KUKA KRL program: MyProgram_017().src

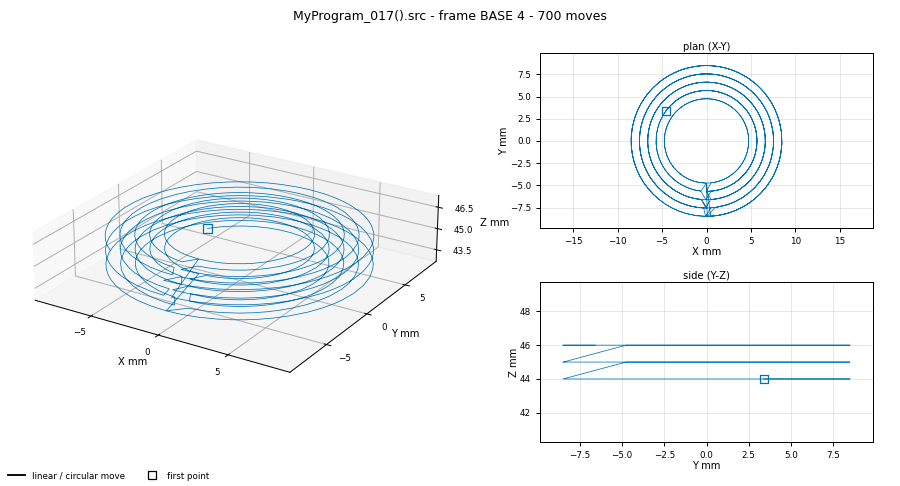
[picture p0: tool path of MyProgram_017().src in frame BASE 4, 700 of 700 moves have a stored position in this frame; points joined in program order, loops and branches not executed]
&ACCESS RVP
&REL 1
&PARAM TEMPLATE = C:\KRC\Roboter\Template\vorgabe
&PARAM EDITMASK = *
DEF MyProgram_017()
; ---- Setting reference (Base) ----
$BASE = BASE_DATA[4]

; --------------------------
; ---- Setting tool (TCP) ----
$TOOL = TOOL_DATA[3]
; --------------------------

$VEL.CP = VEL_APROX_PRINT
Startdeposition()
$VEL.CP = VEL_PRINT
LIN {X -4.5752,Y 3.3749,Z 44,A -2.6957,B 0,C 0,E1 0.1598,E2 90.0717} C_DIS
LIN {X -4.041,Y 3.9987,Z 44,A -2.6496,B 0,C 0,E1 0.1598,E2 90.0718} C_DIS
LIN {X -3.423,Y 4.5393,Z 44,A -2.604,B 0,C 0,E1 0.1598,E2 90.072} C_DIS
LIN {X -2.7335,Y 4.9851,Z 44,A -2.5597,B 0,C 0,E1 0.1598,E2 90.072} C_DIS
LIN {X -1.9869,Y 5.3273,Z 44,A -2.5177,B 0,C 0,E1 0.1598,E2 90.0722} C_DIS
LIN {X -1.1986,Y 5.5572,Z 44,A -2.4789,B 0,C 0,E1 0.1598,E2 90.0722} C_DIS
LIN {X -0.3854,Y 5.6706,Z 44,A -2.4442,B 0,C 0,E1 0.1598,E2 90.0723} C_DIS
LIN {X 0.4354,Y 5.6661,Z 44,A -2.4141,B 0,C 0,E1 0.1598,E2 90.0723} C_DIS
LIN {X 1.247,Y 5.5441,Z 44,A -2.3893,B 0,C 0,E1 0.1598,E2 90.0723} C_DIS
LIN {X 2.0326,Y 5.3067,Z 44,A -2.3704,B 0,C 0,E1 0.1598,E2 90.0723} C_DIS
LIN {X 2.7757,Y 4.9583,Z 44,A -2.3578,B 0,C 0,E1 0.1598,E2 90.0723} C_DIS
LIN {X 3.4609,Y 4.5066,Z 44,A -2.3517,B 0,C 0,E1 0.1598,E2 90.0723} C_DIS
LIN {X 4.0741,Y 3.9612,Z 44,A -2.3522,B 0,C 0,E1 0.1598,E2 90.0723} C_DIS
LIN {X 4.6028,Y 3.3334,Z 44,A -2.3594,B 0,C 0,E1 0.1598,E2 90.0722} C_DIS
LIN {X 5.035,Y 2.6356,Z 44,A -2.3732,B 0,C 0,E1 0.1598,E2 90.0722} C_DIS
LIN {X 5.3636,Y 1.8833,Z 44,A -2.3931,B 0,C 0,E1 0.1598,E2 90.072} C_DIS
LIN {X 5.5801,Y 1.0912,Z 44,A -2.4188,B 0,C 0,E1 0.1598,E2 90.072} C_DIS
LIN {X 5.677,Y 0.2759,Z 44,A -2.45,B 0,C 0,E1 0.1598,E2 90.072} C_DIS
LIN {X 5.6571,Y -0.5447,Z 44,A -2.4857,B 0,C 0,E1 0.1598,E2 90.0719} C_DIS
LIN {X 5.4744,Y -1.5545,Z 44,A -2.5352,B 0,C 0,E1 0.1598,E2 90.0715} C_DIS
LIN {X 5.0638,Y -2.5861,Z 44,A -2.5943,B 0,C 0,E1 0.1598,E2 90.0715} C_DIS
LIN {X 4.6754,Y -3.2361,Z 44,A -2.6367,B 0,C 0,E1 0.1598,E2 90.0718} C_DIS
LIN {X 4.2019,Y -3.8269,Z 44,A -2.6793,B 0,C 0,E1 0.1598,E2 90.0718} C_DIS
LIN {X 3.6555,Y -4.3507,Z 44,A -2.7217,B 0,C 0,E1 0.1598,E2 90.0718} C_DIS
LIN {X 3.0454,Y -4.7986,Z 44,A -2.7633,B 0,C 0,E1 0.1598,E2 90.0718} C_DIS
LIN {X 2.3814,Y -5.1623,Z 44,A -2.8032,B 0,C 0,E1 0.1598,E2 90.0718} C_DIS
LIN {X 1.6745,Y -5.4336,Z 44,A -2.8407,B 0,C 0,E1 0.1598,E2 90.0718} C_DIS
LIN {X 0.9371,Y -5.6051,Z 44,A -2.8751,B 0,C 0,E1 0.1598,E2 90.0718} C_DIS
LIN {X -0.0053,Y -5.6863,Z 44,A -2.9131,B 0,C 0,E1 0.1598,E2 90.0717} C_DIS
Enddeposition()
LIN {X -0.0053,Y -5.6863,Z 44,A -2.9131,B 0,C 0,E1 0.1598,E2 90.0717} C_DIS
Startdeposition()
$VEL.CP = VEL_PRINT
LIN {X 0.5091,Y -6.6003,Z 44,A -2.9327,B 0,C 0,E1 0.1598,E2 90.0711} C_DIS
LIN {X 1.1965,Y -6.5109,Z 44,A -2.9042,B 0,C 0,E1 0.1598,E2 90.0717} C_DIS
LIN {X 1.8711,Y -6.3511,Z 44,A -2.8727,B 0,C 0,E1 0.1598,E2 90.0717} C_DIS
LIN {X 2.5251,Y -6.121,Z 44,A -2.8389,B 0,C 0,E1 0.1598,E2 90.0717} C_DIS
LIN {X 3.1505,Y -5.8217,Z 44,A -2.8032,B 0,C 0,E1 0.1598,E2 90.0717} C_DIS
LIN {X 3.7429,Y -5.4614,Z 44,A -2.7661,B 0,C 0,E1 0.1598,E2 90.0718} C_DIS
LIN {X 4.293,Y -5.0397,Z 44,A -2.7279,B 0,C 0,E1 0.1598,E2 90.0718} C_DIS
LIN {X 4.7982,Y -4.5646,Z 44,A -2.689,B 0,C 0,E1 0.1598,E2 90.0718} C_DIS
LIN {X 5.2469,Y -4.036,Z 44,A -2.65,B 0,C 0,E1 0.1598,E2 90.0718} C_DIS
LIN {X 5.6408,Y -3.4655,Z 44,A -2.6111,B 0,C 0,E1 0.1598,E2 90.0719} C_DIS
LIN {X 5.9718,Y -2.8562,Z 44,A -2.573,B 0,C 0,E1 0.1598,E2 90.0719} C_DIS
LIN {X 6.2393,Y -2.2166,Z 44,A -2.5358,B 0,C 0,E1 0.1598,E2 90.0719} C_DIS
LIN {X 6.4359,Y -1.5516,Z 44,A -2.5002,B 0,C 0,E1 0.1598,E2 90.0719} C_DIS
LIN {X 6.5608,Y -0.8697,Z 44,A -2.4665,B 0,C 0,E1 0.1598,E2 90.072} C_DIS
LIN {X 6.6185,Y -0.1788,Z 44,A -2.4349,B 0,C 0,E1 0.1598,E2 90.072} C_DIS
LIN {X 6.6015,Y 0.5143,Z 44,A -2.4059,B 0,C 0,E1 0.1598,E2 90.072} C_DIS
LIN {X 6.5099,Y 1.2015,Z 44,A -2.38,B 0,C 0,E1 0.1598,E2 90.0721} C_DIS
LIN {X 6.3497,Y 1.876,Z 44,A -2.3571,B 0,C 0,E1 0.1598,E2 90.0721} C_DIS
LIN {X 6.1191,Y 2.5298,Z 44,A -2.3378,B 0,C 0,E1 0.1598,E2 90.0721} C_DIS
LIN {X 5.8214,Y 3.156,Z 44,A -2.3221,B 0,C 0,E1 0.1598,E2 90.0722} C_DIS
LIN {X 5.4565,Y 3.7455,Z 44,A -2.3104,B 0,C 0,E1 0.1598,E2 90.0722} C_DIS
LIN {X 5.0353,Y 4.2961,Z 44,A -2.3025,B 0,C 0,E1 0.1598,E2 90.0723} C_DIS
LIN {X 4.5594,Y 4.8001,Z 44,A -2.2986,B 0,C 0,E1 0.1598,E2 90.0723} C_DIS
LIN {X 4.0329,Y 5.2514,Z 44,A -2.2989,B 0,C 0,E1 0.1598,E2 90.0723} C_DIS
LIN {X 3.461,Y 5.6435,Z 44,A -2.3033,B 0,C 0,E1 0.1598,E2 90.0723} C_DIS
LIN {X 2.8513,Y 5.9736,Z 44,A -2.3118,B 0,C 0,E1 0.1598,E2 90.0724} C_DIS
LIN {X 2.2116,Y 6.2407,Z 44,A -2.324,B 0,C 0,E1 0.1598,E2 90.0724} C_DIS
LIN {X 1.5467,Y 6.4373,Z 44,A -2.3402,B 0,C 0,E1 0.1598,E2 90.0724} C_DIS
LIN {X 0.8651,Y 6.5635,Z 44,A -2.36,B 0,C 0,E1 0.1598,E2 90.0724} C_DIS
LIN {X 0.1739,Y 6.617,Z 44,A -2.3833,B 0,C 0,E1 0.1598,E2 90.0724} C_DIS
LIN {X -0.5191,Y 6.5985,Z 44,A -2.4096,B 0,C 0,E1 0.1598,E2 90.0724} C_DIS
LIN {X -1.2065,Y 6.5086,Z 44,A -2.4388,B 0,C 0,E1 0.1598,E2 90.0724} C_DIS
LIN {X -1.8803,Y 6.3461,Z 44,A -2.4705,B 0,C 0,E1 0.1598,E2 90.0723} C_DIS
LIN {X -2.5337,Y 6.1145,Z 44,A -2.5044,B 0,C 0,E1 0.1598,E2 90.0723} C_DIS
LIN {X -3.1598,Y 5.8167,Z 44,A -2.5401,B 0,C 0,E1 0.1598,E2 90.0721} C_DIS
LIN {X -3.7509,Y 5.4545,Z 44,A -2.5773,B 0,C 0,E1 0.1598,E2 90.0721} C_DIS
LIN {X -4.3009,Y 5.0324,Z 44,A -2.6154,B 0,C 0,E1 0.1598,E2 90.072} C_DIS
LIN {X -4.8047,Y 4.5559,Z 44,A -2.6541,B 0,C 0,E1 0.1598,E2 90.072} C_DIS
LIN {X -5.2547,Y 4.0286,Z 44,A -2.693,B 0,C 0,E1 0.1598,E2 90.0718} C_DIS
LIN {X -5.6466,Y 3.4565,Z 44,A -2.7316,B 0,C 0,E1 0.1598,E2 90.0718} C_DIS
LIN {X -5.9766,Y 2.8467,Z 44,A -2.7695,B 0,C 0,E1 0.1598,E2 90.0717} C_DIS
LIN {X -6.24,Y 2.2054,Z 44,A -2.8064,B 0,C 0,E1 0.1598,E2 90.0717} C_DIS
LIN {X -6.4373,Y 1.5409,Z 44,A -2.8417,B 0,C 0,E1 0.1598,E2 90.0716} C_DIS
LIN {X -6.5877,Y 0.6875,Z 44,A -2.8832,B 0,C 0,E1 0.1598,E2 90.0713} C_DIS
LIN {X -6.6081,Y -0.3658,Z 44,A -2.9284,B 0,C 0,E1 0.1598,E2 90.0711} C_DIS
LIN {X -6.5292,Y -1.09,Z 44,A -2.9564,B 0,C 0,E1 0.1598,E2 90.0713} C_DIS
LIN {X -6.37,Y -1.8008,Z 44,A -2.9807,B 0,C 0,E1 0.1598,E2 90.0713} C_DIS
LIN {X -6.1338,Y -2.49,Z 44,A -3.0013,B 0,C 0,E1 0.1598,E2 90.0713} C_DIS
LIN {X -5.8219,Y -3.1483,Z 44,A -3.0177,B 0,C 0,E1 0.1598,E2 90.0713} C_DIS
LIN {X -5.4419,Y -3.7698,Z 44,A -3.0301,B 0,C 0,E1 0.1598,E2 90.0713} C_DIS
LIN {X -4.9946,Y -4.3449,Z 44,A -3.0381,B 0,C 0,E1 0.1598,E2 90.0713} C_DIS
LIN {X -4.4875,Y -4.8678,Z 44,A -3.0418,B 0,C 0,E1 0.1598,E2 90.0713} C_DIS
LIN {X -3.925,Y -5.3307,Z 44,A -3.0408,B 0,C 0,E1 0.1598,E2 90.0714} C_DIS
LIN {X -3.3151,Y -5.729,Z 44,A -3.0354,B 0,C 0,E1 0.1598,E2 90.0714} C_DIS
LIN {X -2.6657,Y -6.0589,Z 44,A -3.0256,B 0,C 0,E1 0.1598,E2 90.0714} C_DIS
LIN {X -1.9844,Y -6.317,Z 44,A -3.0116,B 0,C 0,E1 0.1598,E2 90.0715} C_DIS
LIN {X -1.2782,Y -6.4958,Z 44,A -2.9933,B 0,C 0,E1 0.1598,E2 90.0715} C_DIS
LIN {X -0.5566,Y -6.5965,Z 44,A -2.9711,B 0,C 0,E1 0.1598,E2 90.0716} C_DIS
LIN {X -0.5566,Y -6.5965,Z 44,A -2.9711,B 0,C 0,E1 0.1598,E2 90.0716} C_DIS
Enddeposition()
LIN {X 0.0479,Y -7.5529,Z 44,A -2.9887,B 0,C 0,E1 0.1598,E2 90.0704} C_DIS
Startdeposition()
$VEL.CP = VEL_PRINT
LIN {X -0.8324,Y -7.5061,Z 44,A -3.0201,B 0,C 0,E1 0.1598,E2 90.0715} C_DIS
LIN {X -1.869,Y -7.322,Z 44,A -3.0503,B 0,C 0,E1 0.1598,E2 90.0715} C_DIS
LIN {X -2.8979,Y -6.9791,Z 44,A -3.0734,B 0,C 0,E1 0.1598,E2 90.0715} C_DIS
LIN {X -3.6656,Y -6.6079,Z 44,A -3.0857,B 0,C 0,E1 0.1598,E2 90.0713} C_DIS
LIN {X -4.6982,Y -5.9194,Z 44,A -3.0942,B 0,C 0,E1 0.1598,E2 90.0713} C_DIS
LIN {X -5.6019,Y -5.0743,Z 44,A -3.0913,B 0,C 0,E1 0.1598,E2 90.071} C_DIS
LIN {X -6.2587,Y -4.232,Z 44,A -3.0797,B 0,C 0,E1 0.1598,E2 90.071} C_DIS
LIN {X -6.6246,Y -3.6273,Z 44,A -3.0677,B 0,C 0,E1 0.1598,E2 90.0713} C_DIS
LIN {X -7.0723,Y -2.6624,Z 44,A -3.043,B 0,C 0,E1 0.1598,E2 90.071} C_DIS
LIN {X -7.3374,Y -1.7971,Z 44,A -3.0162,B 0,C 0,E1 0.1598,E2 90.0712} C_DIS
LIN {X -7.4759,Y -1.0866,Z 44,A -2.9913,B 0,C 0,E1 0.1598,E2 90.0713} C_DIS
LIN {X -7.5584,Y -0.0211,Z 44,A -2.9489,B 0,C 0,E1 0.1598,E2 90.0711} C_DIS
LIN {X -7.4541,Y 1.2425,Z 44,A -2.8914,B 0,C 0,E1 0.1598,E2 90.0709} C_DIS
LIN {X -7.1635,Y 2.3945,Z 44,A -2.832,B 0,C 0,E1 0.1598,E2 90.071} C_DIS
LIN {X -6.6973,Y 3.5029,Z 44,A -2.7681,B 0,C 0,E1 0.1598,E2 90.0713} C_DIS
LIN {X -6.1734,Y 4.3532,Z 44,A -2.7131,B 0,C 0,E1 0.1598,E2 90.0716} C_DIS
LIN {X -5.6769,Y 4.9792,Z 44,A -2.6684,B 0,C 0,E1 0.1598,E2 90.0718} C_DIS
LIN {X -4.9743,Y 5.6888,Z 44,A -2.6124,B 0,C 0,E1 0.1598,E2 90.0718} C_DIS
LIN {X -4.1104,Y 6.3399,Z 44,A -2.553,B 0,C 0,E1 0.1598,E2 90.072} C_DIS
LIN {X -3.0954,Y 6.8952,Z 44,A -2.4921,B 0,C 0,E1 0.1598,E2 90.072} C_DIS
LIN {X -1.8698,Y 7.3218,Z 44,A -2.4289,B 0,C 0,E1 0.1598,E2 90.0722} C_DIS
LIN {X -0.7337,Y 7.5179,Z 44,A -2.3787,B 0,C 0,E1 0.1598,E2 90.0724} C_DIS
LIN {X 0.0199,Y 7.5584,Z 44,A -2.3492,B 0,C 0,E1 0.1598,E2 90.0724} C_DIS
LIN {X 1.0346,Y 7.4814,Z 44,A -2.315,B 0,C 0,E1 0.1598,E2 90.0724} C_DIS
LIN {X 2.3327,Y 7.188,Z 44,A -2.2795,B 0,C 0,E1 0.1598,E2 90.0724} C_DIS
LIN {X 3.4366,Y 6.7315,Z 44,A -2.2581,B 0,C 0,E1 0.1598,E2 90.0724} C_DIS
LIN {X 4.3592,Y 6.1685,Z 44,A -2.2479,B 0,C 0,E1 0.1598,E2 90.0724} C_DIS
LIN {X 4.9311,Y 5.7235,Z 44,A -2.2459,B 0,C 0,E1 0.1598,E2 90.0724} C_DIS
LIN {X 5.703,Y 4.9577,Z 44,A -2.2498,B 0,C 0,E1 0.1598,E2 90.0722} C_DIS
LIN {X 6.1582,Y 4.3734,Z 44,A -2.258,B 0,C 0,E1 0.1598,E2 90.0722} C_DIS
LIN {X 6.5699,Y 3.7348,Z 44,A -2.2699,B 0,C 0,E1 0.1598,E2 90.0722} C_DIS
LIN {X 6.951,Y 2.9639,Z 44,A -2.2888,B 0,C 0,E1 0.1598,E2 90.0722} C_DIS
LIN {X 7.3186,Y 1.8702,Z 44,A -2.3214,B 0,C 0,E1 0.1598,E2 90.0717} C_DIS
LIN {X 7.5125,Y 0.8179,Z 44,A -2.3592,B 0,C 0,E1 0.1598,E2 90.0717} C_DIS
LIN {X 7.5542,Y -0.2068,Z 44,A -2.4015,B 0,C 0,E1 0.1598,E2 90.0717} C_DIS
LIN {X 7.4289,Y -1.3641,Z 44,A -2.4555,B 0,C 0,E1 0.1598,E2 90.0717} C_DIS
LIN {X 7.1177,Y -2.5389,Z 44,A -2.517,B 0,C 0,E1 0.1598,E2 90.0715} C_DIS
LIN {X 6.8077,Y -3.2797,Z 44,A -2.5603,B 0,C 0,E1 0.1598,E2 90.0718} C_DIS
LIN {X 6.3045,Y -4.1586,Z 44,A -2.6163,B 0,C 0,E1 0.1598,E2 90.0718} C_DIS
LIN {X 5.8221,Y -4.8095,Z 44,A -2.662,B 0,C 0,E1 0.1598,E2 90.0718} C_DIS
LIN {X 5.2731,Y -5.4052,Z 44,A -2.7076,B 0,C 0,E1 0.1598,E2 90.0718} C_DIS
LIN {X 4.6638,Y -5.9391,Z 44,A -2.7528,B 0,C 0,E1 0.1598,E2 90.0718} C_DIS
LIN {X 4.0007,Y -6.4044,Z 44,A -2.797,B 0,C 0,E1 0.1598,E2 90.0718} C_DIS
LIN {X 3.0197,Y -6.9273,Z 44,A -2.8552,B 0,C 0,E1 0.1598,E2 90.0716} C_DIS
LIN {X 2.2786,Y -7.2008,Z 44,A -2.8941,B 0,C 0,E1 0.1598,E2 90.0716} C_DIS
LIN {X 0.9731,Y -7.4949,Z 44,A -2.9545,B 0,C 0,E1 0.1598,E2 90.0716} C_DIS
LIN {X 0.9731,Y -7.4949,Z 44,A -2.9545,B 0,C 0,E1 0.1598,E2 90.0716} C_DIS
Enddeposition()
LIN {X 0.0783,Y -8.4906,Z 44,A -3.0288,B 0,C 0,E1 0.1598,E2 90.0703} C_DIS
Startdeposition()
$VEL.CP = VEL_PRINT
LIN {X 1.1261,Y -8.4125,Z 44,A -2.9882,B 0,C 0,E1 0.1598,E2 90.0715} C_DIS
LIN {X 2.1575,Y -8.2116,Z 44,A -2.9419,B 0,C 0,E1 0.1598,E2 90.0716} C_DIS
LIN {X 3.3011,Y -7.8174,Z 44,A -2.8831,B 0,C 0,E1 0.1598,E2 90.0716} C_DIS
LIN {X 4.0529,Y -7.4557,Z 44,A -2.8401,B 0,C 0,E1 0.1598,E2 90.0717} C_DIS
LIN {X 4.7655,Y -7.0219,Z 44,A -2.7954,B 0,C 0,E1 0.1598,E2 90.0717} C_DIS
LIN {X 5.4321,Y -6.5202,Z 44,A -2.7496,B 0,C 0,E1 0.1598,E2 90.0717} C_DIS
LIN {X 6.0464,Y -5.9555,Z 44,A -2.7029,B 0,C 0,E1 0.1598,E2 90.0718} C_DIS
LIN {X 6.7336,Y -5.171,Z 44,A -2.6439,B 0,C 0,E1 0.1598,E2 90.0717} C_DIS
LIN {X 7.4358,Y -4.0976,Z 44,A -2.572,B 0,C 0,E1 0.1598,E2 90.0715} C_DIS
LIN {X 7.8887,Y -3.1313,Z 44,A -2.5143,B 0,C 0,E1 0.1598,E2 90.0717} C_DIS
LIN {X 8.1635,Y -2.3229,Z 44,A -2.4698,B 0,C 0,E1 0.1598,E2 90.0719} C_DIS
LIN {X 8.3559,Y -1.491,Z 44,A -2.4271,B 0,C 0,E1 0.1598,E2 90.0719} C_DIS
LIN {X 8.4854,Y -0.3279,Z 44,A -2.3724,B 0,C 0,E1 0.1598,E2 90.0717} C_DIS
LIN {X 8.4327,Y 0.9895,Z 44,A -2.3179,B 0,C 0,E1 0.1598,E2 90.0716} C_DIS
LIN {X 8.1637,Y 2.339,Z 44,A -2.27,B 0,C 0,E1 0.1598,E2 90.0715} C_DIS
LIN {X 7.7132,Y 3.5398,Z 44,A -2.2355,B 0,C 0,E1 0.1598,E2 90.0716} C_DIS
LIN {X 7.3654,Y 4.2257,Z 44,A -2.2195,B 0,C 0,E1 0.1598,E2 90.0722} C_DIS
LIN {X 6.789,Y 5.0922,Z 44,A -2.2039,B 0,C 0,E1 0.1598,E2 90.0722} C_DIS
LIN {X 6.2576,Y 5.7333,Z 44,A -2.1963,B 0,C 0,E1 0.1598,E2 90.0724} C_DIS
LIN {X 5.5108,Y 6.4584,Z 44,A -2.1929,B 0,C 0,E1 0.1598,E2 90.0723} C_DIS
LIN {X 4.4748,Y 7.2151,Z 44,A -2.1989,B 0,C 0,E1 0.1598,E2 90.0723} C_DIS
LIN {X 3.4884,Y 7.7361,Z 44,A -2.2133,B 0,C 0,E1 0.1598,E2 90.0724} C_DIS
LIN {X 2.6566,Y 8.0595,Z 44,A -2.2304,B 0,C 0,E1 0.1598,E2 90.0725} C_DIS
LIN {X 1.7956,Y 8.2944,Z 44,A -2.2522,B 0,C 0,E1 0.1598,E2 90.0725} C_DIS
LIN {X 0.9149,Y 8.4383,Z 44,A -2.2787,B 0,C 0,E1 0.1598,E2 90.0725} C_DIS
LIN {X -0.1995,Y 8.4882,Z 44,A -2.3177,B 0,C 0,E1 0.1598,E2 90.0725} C_DIS
LIN {X -1.2766,Y 8.3942,Z 44,A -2.3615,B 0,C 0,E1 0.1598,E2 90.0725} C_DIS
LIN {X -2.3519,Y 8.1545,Z 44,A -2.4113,B 0,C 0,E1 0.1598,E2 90.0723} C_DIS
LIN {X -3.1851,Y 7.8669,Z 44,A -2.4542,B 0,C 0,E1 0.1598,E2 90.0723} C_DIS
LIN {X -3.9839,Y 7.4946,Z 44,A -2.4994,B 0,C 0,E1 0.1598,E2 90.0722} C_DIS
LIN {X -4.7396,Y 7.0409,Z 44,A -2.5465,B 0,C 0,E1 0.1598,E2 90.0721} C_DIS
LIN {X -5.4443,Y 6.5115,Z 44,A -2.5949,B 0,C 0,E1 0.1598,E2 90.072} C_DIS
LIN {X -6.3196,Y 5.6726,Z 44,A -2.6624,B 0,C 0,E1 0.1598,E2 90.0717} C_DIS
LIN {X -7.0513,Y 4.7231,Z 44,A -2.7294,B 0,C 0,E1 0.1598,E2 90.0714} C_DIS
LIN {X -7.5,Y 3.9716,Z 44,A -2.7779,B 0,C 0,E1 0.1598,E2 90.0716} C_DIS
LIN {X -7.8689,Y 3.1778,Z 44,A -2.825,B 0,C 0,E1 0.1598,E2 90.0715} C_DIS
LIN {X -8.1548,Y 2.3506,Z 44,A -2.8705,B 0,C 0,E1 0.1598,E2 90.0714} C_DIS
LIN {X -8.3541,Y 1.4983,Z 44,A -2.9138,B 0,C 0,E1 0.1598,E2 90.0714} C_DIS
LIN {X -8.4869,Y 0.2593,Z 44,A -2.9707,B 0,C 0,E1 0.1598,E2 90.0709} C_DIS
LIN {X -8.4482,Y -0.8008,Z 44,A -3.0143,B 0,C 0,E1 0.1598,E2 90.071} C_DIS
LIN {X -8.3257,Y -1.6406,Z 44,A -3.0455,B 0,C 0,E1 0.1598,E2 90.0711} C_DIS
LIN {X -8.1203,Y -2.4641,Z 44,A -3.0729,B 0,C 0,E1 0.1598,E2 90.0711} C_DIS
LIN {X -7.8332,Y -3.2627,Z 44,A -3.0961,B 0,C 0,E1 0.1598,E2 90.0711} C_DIS
LIN {X -7.4686,Y -4.0291,Z 44,A -3.1152,B 0,C 0,E1 0.1598,E2 90.0711} C_DIS
LIN {X -7.0291,Y -4.7552,Z 44,A -3.1299,B 0,C 0,E1 0.1598,E2 90.0711} C_DIS
LIN {X -6.5186,Y -5.4333,Z 44,A -3.14,B 0,C 0,E1 0.1598,E2 90.0711} C_DIS
LIN {X -5.9432,Y -6.0572,Z 44,A -3.1453,B 0,C 0,E1 0.1598,E2 90.0711} C_DIS
LIN {X -5.3091,Y -6.6214,Z 44,A -3.1461,B 0,C 0,E1 0.1598,E2 90.0712} C_DIS
LIN {X -4.6211,Y -7.1185,Z 44,A -3.142,B 0,C 0,E1 0.1598,E2 90.0712} C_DIS
LIN {X -3.887,Y -7.5447,Z 44,A -3.1332,B 0,C 0,E1 0.1598,E2 90.0712} C_DIS
LIN {X -3.114,Y -7.8955,Z 44,A -3.1198,B 0,C 0,E1 0.1598,E2 90.0713} C_DIS
LIN {X -2.3098,Y -8.1673,Z 44,A -3.1019,B 0,C 0,E1 0.1598,E2 90.0713} C_DIS
LIN {X -1.1138,Y -8.4185,Z 44,A -3.0688,B 0,C 0,E1 0.1598,E2 90.0714} C_DIS
LIN {X 0.0783,Y -8.4906,Z 44,A -3.0282,B 0,C 0,E1 0.1598,E2 90.0715} C_DIS
Enddeposition()
LIN {X 0.0009,Y -4.7545,Z 45,A -2.8574,B 0,C 0,E1 0.1598,E2 90.0604} C_DIS
Startdeposition()
$VEL.CP = VEL_PRINT
LIN {X 0.0009,Y -4.7545,Z 45,A -2.8631,B 0,C 0,E1 0.1598,E2 90.0661} C_DIS
LIN {X -0.8429,Y -4.6775,Z 45,A -2.8957,B 0,C 0,E1 0.1598,E2 90.071} C_DIS
LIN {X -1.5,Y -4.5101,Z 45,A -2.9134,B 0,C 0,E1 0.1598,E2 90.0716} C_DIS
LIN {X -2.1259,Y -4.2496,Z 45,A -2.9253,B 0,C 0,E1 0.1598,E2 90.0716} C_DIS
LIN {X -2.7086,Y -3.9031,Z 45,A -2.9319,B 0,C 0,E1 0.1598,E2 90.0716} C_DIS
LIN {X -3.2363,Y -3.4777,Z 45,A -2.9332,B 0,C 0,E1 0.1598,E2 90.0716} C_DIS
LIN {X -3.698,Y -2.9814,Z 45,A -2.929,B 0,C 0,E1 0.1598,E2 90.0716} C_DIS
LIN {X -4.0839,Y -2.4243,Z 45,A -2.9195,B 0,C 0,E1 0.1598,E2 90.0716} C_DIS
LIN {X -4.39,Y -1.8195,Z 45,A -2.9051,B 0,C 0,E1 0.1598,E2 90.0715} C_DIS
LIN {X -4.6025,Y -1.1756,Z 45,A -2.8856,B 0,C 0,E1 0.1598,E2 90.0715} C_DIS
LIN {X -4.722,Y -0.5086,Z 45,A -2.8617,B 0,C 0,E1 0.1598,E2 90.0715} C_DIS
LIN {X -4.7473,Y 0.1687,Z 45,A -2.8339,B 0,C 0,E1 0.1598,E2 90.0715} C_DIS
LIN {X -4.677,Y 0.8429,Z 45,A -2.8027,B 0,C 0,E1 0.1598,E2 90.0715} C_DIS
LIN {X -4.4794,Y 1.5793,Z 45,A -2.7642,B 0,C 0,E1 0.1598,E2 90.0715} C_DIS
LIN {X -4.2478,Y 2.1254,Z 45,A -2.7326,B 0,C 0,E1 0.1598,E2 90.0718} C_DIS
LIN {X -3.9031,Y 2.7089,Z 45,A -2.6952,B 0,C 0,E1 0.1598,E2 90.0718} C_DIS
LIN {X -3.4776,Y 3.2366,Z 45,A -2.6572,B 0,C 0,E1 0.1598,E2 90.0718} C_DIS
LIN {X -2.9811,Y 3.6982,Z 45,A -2.6194,B 0,C 0,E1 0.1598,E2 90.072} C_DIS
LIN {X -2.4244,Y 4.0846,Z 45,A -2.5825,B 0,C 0,E1 0.1598,E2 90.072} C_DIS
LIN {X -1.8183,Y 4.3878,Z 45,A -2.5473,B 0,C 0,E1 0.1598,E2 90.0721} C_DIS
LIN {X -1.1756,Y 4.6029,Z 45,A -2.5145,B 0,C 0,E1 0.1598,E2 90.0721} C_DIS
LIN {X -0.5087,Y 4.7244,Z 45,A -2.4848,B 0,C 0,E1 0.1598,E2 90.0723} C_DIS
LIN {X 0.1688,Y 4.7487,Z 45,A -2.4588,B 0,C 0,E1 0.1598,E2 90.0723} C_DIS
LIN {X 0.8431,Y 4.6778,Z 45,A -2.437,B 0,C 0,E1 0.1598,E2 90.0723} C_DIS
LIN {X 1.5,Y 4.5098,Z 45,A -2.4199,B 0,C 0,E1 0.1598,E2 90.0723} C_DIS
LIN {X 2.1262,Y 4.2496,Z 45,A -2.4078,B 0,C 0,E1 0.1598,E2 90.0723} C_DIS
LIN {X 2.7087,Y 3.9029,Z 45,A -2.4011,B 0,C 0,E1 0.1598,E2 90.0723} C_DIS
LIN {X 3.2365,Y 3.4775,Z 45,A -2.3997,B 0,C 0,E1 0.1598,E2 90.0723} C_DIS
LIN {X 3.6981,Y 2.9812,Z 45,A -2.4038,B 0,C 0,E1 0.1598,E2 90.0723} C_DIS
LIN {X 4.085,Y 2.4247,Z 45,A -2.4132,B 0,C 0,E1 0.1598,E2 90.0722} C_DIS
LIN {X 4.3887,Y 1.8188,Z 45,A -2.4278,B 0,C 0,E1 0.1598,E2 90.0722} C_DIS
LIN {X 4.6034,Y 1.1759,Z 45,A -2.4472,B 0,C 0,E1 0.1598,E2 90.0721} C_DIS
LIN {X 4.7244,Y 0.5089,Z 45,A -2.4712,B 0,C 0,E1 0.1598,E2 90.0721} C_DIS
LIN {X 4.746,Y -0.1685,Z 45,A -2.4992,B 0,C 0,E1 0.1598,E2 90.072} C_DIS
LIN {X 4.6768,Y -0.8428,Z 45,A -2.5305,B 0,C 0,E1 0.1598,E2 90.072} C_DIS
LIN {X 4.5095,Y -1.4998,Z 45,A -2.5647,B 0,C 0,E1 0.1598,E2 90.072} C_DIS
LIN {X 4.2493,Y -2.1258,Z 45,A -2.601,B 0,C 0,E1 0.1598,E2 90.0719} C_DIS
LIN {X 3.9024,Y -2.7081,Z 45,A -2.6386,B 0,C 0,E1 0.1598,E2 90.0719} C_DIS
LIN {X 3.4789,Y -3.2377,Z 45,A -2.6767,B 0,C 0,E1 0.1598,E2 90.0719} C_DIS
LIN {X 2.982,Y -3.6988,Z 45,A -2.7147,B 0,C 0,E1 0.1598,E2 90.0719} C_DIS
LIN {X 2.4254,Y -4.086,Z 45,A -2.7516,B 0,C 0,E1 0.1598,E2 90.0719} C_DIS
LIN {X 1.8183,Y -4.3879,Z 45,A -2.7868,B 0,C 0,E1 0.1598,E2 90.0719} C_DIS
LIN {X 1.1758,Y -4.6031,Z 45,A -2.8196,B 0,C 0,E1 0.1598,E2 90.0718} C_DIS
LIN {X 0.5088,Y -4.7245,Z 45,A -2.8492,B 0,C 0,E1 0.1598,E2 90.0718} C_DIS
LIN {X 0.5088,Y -4.7245,Z 45,A -2.8492,B 0,C 0,E1 0.1598,E2 90.0718} C_DIS
Enddeposition()
LIN {X -0.0394,Y -5.6894,Z 45,A -2.9094,B 0,C 0,E1 0.1598,E2 90.0705} C_DIS
Startdeposition()
$VEL.CP = VEL_PRINT
LIN {X 0.9442,Y -5.6043,Z 45,A -2.8708,B 0,C 0,E1 0.1598,E2 90.0717} C_DIS
LIN {X 1.7118,Y -5.4187,Z 45,A -2.8348,B 0,C 0,E1 0.1598,E2 90.0717} C_DIS
LIN {X 2.4465,Y -5.1294,Z 45,A -2.7954,B 0,C 0,E1 0.1598,E2 90.0718} C_DIS
LIN {X 3.1348,Y -4.7418,Z 45,A -2.7536,B 0,C 0,E1 0.1598,E2 90.0718} C_DIS
LIN {X 3.7623,Y -4.2619,Z 45,A -2.7101,B 0,C 0,E1 0.1598,E2 90.0718} C_DIS
LIN {X 4.4468,Y -3.55,Z 45,A -2.6544,B 0,C 0,E1 0.1598,E2 90.0718} C_DIS
LIN {X 5.0417,Y -2.6289,Z 45,A -2.5931,B 0,C 0,E1 0.1598,E2 90.0716} C_DIS
LIN {X 5.3446,Y -1.9384,Z 45,A -2.5527,B 0,C 0,E1 0.1598,E2 90.0719} C_DIS
LIN {X 5.5518,Y -1.2134,Z 45,A -2.5142,B 0,C 0,E1 0.1598,E2 90.0719} C_DIS
LIN {X 5.688,Y -0.1413,Z 45,A -2.4631,B 0,C 0,E1 0.1598,E2 90.0717} C_DIS
LIN {X 5.6672,Y 0.4603,Z 45,A -2.4385,B 0,C 0,E1 0.1598,E2 90.072} C_DIS
LIN {X 5.5456,Y 1.2531,Z 45,A -2.4091,B 0,C 0,E1 0.1598,E2 90.072} C_DIS
LIN {X 5.3129,Y 2.0206,Z 45,A -2.385,B 0,C 0,E1 0.1598,E2 90.072} C_DIS
LIN {X 4.9742,Y 2.7475,Z 45,A -2.3665,B 0,C 0,E1 0.1598,E2 90.0721} C_DIS
LIN {X 4.5374,Y 3.4198,Z 45,A -2.354,B 0,C 0,E1 0.1598,E2 90.0721} C_DIS
LIN {X 4.0116,Y 4.025,Z 45,A -2.3477,B 0,C 0,E1 0.1598,E2 90.0722} C_DIS
LIN {X 3.4053,Y 4.5498,Z 45,A -2.3477,B 0,C 0,E1 0.1598,E2 90.0722} C_DIS
LIN {X 2.7307,Y 4.9828,Z 45,A -2.3542,B 0,C 0,E1 0.1598,E2 90.0723} C_DIS
LIN {X 2.0026,Y 5.3184,Z 45,A -2.3669,B 0,C 0,E1 0.1598,E2 90.0723} C_DIS
LIN {X 1.2344,Y 5.5481,Z 45,A -2.3855,B 0,C 0,E1 0.1598,E2 90.0723} C_DIS
LIN {X 0.4413,Y 5.6676,Z 45,A -2.4097,B 0,C 0,E1 0.1598,E2 90.0723} C_DIS
LIN {X -0.3607,Y 5.6737,Z 45,A -2.439,B 0,C 0,E1 0.1598,E2 90.0723} C_DIS
LIN {X -1.1555,Y 5.5658,Z 45,A -2.4729,B 0,C 0,E1 0.1598,E2 90.0723} C_DIS
LIN {X -1.927,Y 5.3469,Z 45,A -2.5106,B 0,C 0,E1 0.1598,E2 90.0723} C_DIS
LIN {X -2.6598,Y 5.0216,Z 45,A -2.5514,B 0,C 0,E1 0.1598,E2 90.0721} C_DIS
LIN {X -3.34,Y 4.5972,Z 45,A -2.5944,B 0,C 0,E1 0.1598,E2 90.0721} C_DIS
LIN {X -3.9536,Y 4.0813,Z 45,A -2.6388,B 0,C 0,E1 0.1598,E2 90.0719} C_DIS
LIN {X -4.4898,Y 3.4851,Z 45,A -2.6838,B 0,C 0,E1 0.1598,E2 90.0719} C_DIS
LIN {X -4.9352,Y 2.8183,Z 45,A -2.7284,B 0,C 0,E1 0.1598,E2 90.0717} C_DIS
LIN {X -5.2826,Y 2.0957,Z 45,A -2.7717,B 0,C 0,E1 0.1598,E2 90.0717} C_DIS
LIN {X -5.5242,Y 1.3312,Z 45,A -2.813,B 0,C 0,E1 0.1598,E2 90.0715} C_DIS
LIN {X -5.6578,Y 0.5406,Z 45,A -2.8514,B 0,C 0,E1 0.1598,E2 90.0715} C_DIS
LIN {X -5.6767,Y -0.261,Z 45,A -2.886,B 0,C 0,E1 0.1598,E2 90.0714} C_DIS
LIN {X -5.5834,Y -1.0572,Z 45,A -2.9163,B 0,C 0,E1 0.1598,E2 90.0714} C_DIS
LIN {X -5.3808,Y -1.8331,Z 45,A -2.9418,B 0,C 0,E1 0.1598,E2 90.0714} C_DIS
LIN {X -5.0704,Y -2.5726,Z 45,A -2.9617,B 0,C 0,E1 0.1598,E2 90.0714} C_DIS
LIN {X -4.6577,Y -3.2604,Z 45,A -2.9758,B 0,C 0,E1 0.1598,E2 90.0714} C_DIS
LIN {X -4.1521,Y -3.8833,Z 45,A -2.9837,B 0,C 0,E1 0.1598,E2 90.0714} C_DIS
LIN {X -3.5643,Y -4.429,Z 45,A -2.9854,B 0,C 0,E1 0.1598,E2 90.0714} C_DIS
LIN {X -2.9043,Y -4.8845,Z 45,A -2.9805,B 0,C 0,E1 0.1598,E2 90.0714} C_DIS
LIN {X -2.1875,Y -5.2436,Z 45,A -2.9695,B 0,C 0,E1 0.1598,E2 90.0715} C_DIS
LIN {X -1.4289,Y -5.5038,Z 45,A -2.9528,B 0,C 0,E1 0.1598,E2 90.0715} C_DIS
LIN {X -0.6401,Y -5.6487,Z 45,A -2.93,B 0,C 0,E1 0.1598,E2 90.0717} C_DIS
LIN {X -0.6401,Y -5.6487,Z 45,A -2.93,B 0,C 0,E1 0.1598,E2 90.0717} C_DIS
Enddeposition()
LIN {X -0.0671,Y -6.6202,Z 45,A -2.9493,B 0,C 0,E1 0.1598,E2 90.0704} C_DIS
Startdeposition()
$VEL.CP = VEL_PRINT
LIN {X -0.9307,Y -6.5542,Z 45,A -2.9793,B 0,C 0,E1 0.1598,E2 90.0715} C_DIS
LIN {X -1.6109,Y -6.4226,Z 45,A -2.9987,B 0,C 0,E1 0.1598,E2 90.0715} C_DIS
LIN {X -2.2736,Y -6.2199,Z 45,A -3.0144,B 0,C 0,E1 0.1598,E2 90.0715} C_DIS
LIN {X -2.9107,Y -5.9471,Z 45,A -3.0261,B 0,C 0,E1 0.1598,E2 90.0715} C_DIS
LIN {X -3.5158,Y -5.6093,Z 45,A -3.034,B 0,C 0,E1 0.1598,E2 90.0715} C_DIS
LIN {X -4.0831,Y -5.2114,Z 45,A -3.0379,B 0,C 0,E1 0.1598,E2 90.0715} C_DIS
LIN {X -4.6042,Y -4.7548,Z 45,A -3.0376,B 0,C 0,E1 0.1598,E2 90.0715} C_DIS
LIN {X -5.0766,Y -4.2479,Z 45,A -3.0334,B 0,C 0,E1 0.1598,E2 90.0714} C_DIS
LIN {X -5.4921,Y -3.6935,Z 45,A -3.0251,B 0,C 0,E1 0.1598,E2 90.0714} C_DIS
LIN {X -5.8502,Y -3.1003,Z 45,A -3.0131,B 0,C 0,E1 0.1598,E2 90.0714} C_DIS
LIN {X -6.1417,Y -2.4717,Z 45,A -2.9971,B 0,C 0,E1 0.1598,E2 90.0714} C_DIS
LIN {X -6.3666,Y -1.8163,Z 45,A -2.9776,B 0,C 0,E1 0.1598,E2 90.0714} C_DIS
LIN {X -6.522,Y -1.141,Z 45,A -2.9546,B 0,C 0,E1 0.1598,E2 90.0714} C_DIS
LIN {X -6.6026,Y -0.4529,Z 45,A -2.9284,B 0,C 0,E1 0.1598,E2 90.0714} C_DIS
LIN {X -6.6158,Y 0.2398,Z 45,A -2.8996,B 0,C 0,E1 0.1598,E2 90.0714} C_DIS
LIN {X -6.5527,Y 0.9298,Z 45,A -2.868,B 0,C 0,E1 0.1598,E2 90.0714} C_DIS
LIN {X -6.4214,Y 1.6102,Z 45,A -2.8344,B 0,C 0,E1 0.1598,E2 90.0715} C_DIS
LIN {X -6.2159,Y 2.2719,Z 45,A -2.7988,B 0,C 0,E1 0.1598,E2 90.0716} C_DIS
LIN {X -5.9449,Y 2.9096,Z 45,A -2.7619,B 0,C 0,E1 0.1598,E2 90.0716} C_DIS
LIN {X -5.609,Y 3.5156,Z 45,A -2.7239,B 0,C 0,E1 0.1598,E2 90.0717} C_DIS
LIN {X -5.2114,Y 4.0831,Z 45,A -2.6852,B 0,C 0,E1 0.1598,E2 90.0718} C_DIS
LIN {X -4.7561,Y 4.6054,Z 45,A -2.6463,B 0,C 0,E1 0.1598,E2 90.0719} C_DIS
LIN {X -4.2479,Y 5.0765,Z 45,A -2.6077,B 0,C 0,E1 0.1598,E2 90.0719} C_DIS
LIN {X -3.6942,Y 5.493,Z 45,A -2.5697,B 0,C 0,E1 0.1598,E2 90.0721} C_DIS
LIN {X -3.099,Y 5.8479,Z 45,A -2.5327,B 0,C 0,E1 0.1598,E2 90.0721} C_DIS
LIN {X -2.4708,Y 6.1401,Z 45,A -2.4972,B 0,C 0,E1 0.1598,E2 90.0722} C_DIS
LIN {X -1.8157,Y 6.3661,Z 45,A -2.4634,B 0,C 0,E1 0.1598,E2 90.0722} C_DIS
LIN {X -1.1405,Y 6.522,Z 45,A -2.4319,B 0,C 0,E1 0.1598,E2 90.0723} C_DIS
LIN {X -0.4526,Y 6.6067,Z 45,A -2.403,B 0,C 0,E1 0.1598,E2 90.0723} C_DIS
LIN {X 0.2403,Y 6.6158,Z 45,A -2.377,B 0,C 0,E1 0.1598,E2 90.0723} C_DIS
LIN {X 0.9305,Y 6.5548,Z 45,A -2.3541,B 0,C 0,E1 0.1598,E2 90.0724} C_DIS
LIN {X 1.6107,Y 6.4225,Z 45,A -2.3347,B 0,C 0,E1 0.1598,E2 90.0724} C_DIS
LIN {X 2.2731,Y 6.219,Z 45,A -2.3188,B 0,C 0,E1 0.1598,E2 90.0724} C_DIS
LIN {X 2.9094,Y 5.9446,Z 45,A -2.307,B 0,C 0,E1 0.1598,E2 90.0724} C_DIS
LIN {X 3.5153,Y 5.6084,Z 45,A -2.299,B 0,C 0,E1 0.1598,E2 90.0724} C_DIS
LIN {X 4.082,Y 5.2097,Z 45,A -2.295,B 0,C 0,E1 0.1598,E2 90.0724} C_DIS
LIN {X 4.6044,Y 4.7545,Z 45,A -2.295,B 0,C 0,E1 0.1598,E2 90.0724} C_DIS
LIN {X 5.0758,Y 4.2468,Z 45,A -2.2993,B 0,C 0,E1 0.1598,E2 90.0724} C_DIS
LIN {X 5.4936,Y 3.694,Z 45,A -2.3074,B 0,C 0,E1 0.1598,E2 90.0724} C_DIS
LIN {X 5.8501,Y 3.0999,Z 45,A -2.3196,B 0,C 0,E1 0.1598,E2 90.0723} C_DIS
LIN {X 6.1414,Y 2.4712,Z 45,A -2.3356,B 0,C 0,E1 0.1598,E2 90.0723} C_DIS
LIN {X 6.3658,Y 1.8155,Z 45,A -2.3553,B 0,C 0,E1 0.1598,E2 90.0722} C_DIS
LIN {X 6.5218,Y 1.1403,Z 45,A -2.3783,B 0,C 0,E1 0.1598,E2 90.0722} C_DIS
LIN {X 6.6053,Y 0.4525,Z 45,A -2.4046,B 0,C 0,E1 0.1598,E2 90.0721} C_DIS
LIN {X 6.6147,Y -0.2405,Z 45,A -2.4338,B 0,C 0,E1 0.1598,E2 90.0721} C_DIS
LIN {X 6.5532,Y -0.9305,Z 45,A -2.4655,B 0,C 0,E1 0.1598,E2 90.0721} C_DIS
LIN {X 6.4206,Y -1.6106,Z 45,A -2.4994,B 0,C 0,E1 0.1598,E2 90.072} C_DIS
LIN {X 6.2178,Y -2.2732,Z 45,A -2.5351,B 0,C 0,E1 0.1598,E2 90.072} C_DIS
LIN {X 5.945,Y -2.9102,Z 45,A -2.5724,B 0,C 0,E1 0.1598,E2 90.072} C_DIS
LIN {X 5.6087,Y -3.516,Z 45,A -2.6106,B 0,C 0,E1 0.1598,E2 90.0719} C_DIS
LIN {X 5.21,Y -4.0827,Z 45,A -2.6494,B 0,C 0,E1 0.1598,E2 90.0719} C_DIS
LIN {X 4.7563,Y -4.6065,Z 45,A -2.6885,B 0,C 0,E1 0.1598,E2 90.0719} C_DIS
LIN {X 4.2476,Y -5.077,Z 45,A -2.7272,B 0,C 0,E1 0.1598,E2 90.0719} C_DIS
LIN {X 3.6941,Y -5.4937,Z 45,A -2.7653,B 0,C 0,E1 0.1598,E2 90.0719} C_DIS
LIN {X 3.0991,Y -5.8489,Z 45,A -2.8023,B 0,C 0,E1 0.1598,E2 90.0718} C_DIS
LIN {X 2.4714,Y -6.1422,Z 45,A -2.8379,B 0,C 0,E1 0.1598,E2 90.0718} C_DIS
LIN {X 1.816,Y -6.3669,Z 45,A -2.8715,B 0,C 0,E1 0.1598,E2 90.0718} C_DIS
LIN {X 1.1405,Y -6.5218,Z 45,A -2.9029,B 0,C 0,E1 0.1598,E2 90.0717} C_DIS
LIN {X 0.4524,Y -6.6029,Z 45,A -2.9316,B 0,C 0,E1 0.1598,E2 90.0717} C_DIS
LIN {X 0.4524,Y -6.6029,Z 45,A -2.9316,B 0,C 0,E1 0.1598,E2 90.0717} C_DIS
Enddeposition()
LIN {X -0.0833,Y -7.5558,Z 45,A -2.9908,B 0,C 0,E1 0.1598,E2 90.0704} C_DIS
Startdeposition()
$VEL.CP = VEL_PRINT
LIN {X 0.9744,Y -7.4948,Z 45,A -2.9506,B 0,C 0,E1 0.1598,E2 90.0716} C_DIS
LIN {X 2.3891,Y -7.1658,Z 45,A -2.8847,B 0,C 0,E1 0.1598,E2 90.0716} C_DIS
LIN {X 3.116,Y -6.8801,Z 45,A -2.8459,B 0,C 0,E1 0.1598,E2 90.0717} C_DIS
LIN {X 4.084,Y -6.3591,Z 45,A -2.7881,B 0,C 0,E1 0.1598,E2 90.0717} C_DIS
LIN {X 4.8796,Y -5.7671,Z 45,A -2.7336,B 0,C 0,E1 0.1598,E2 90.0717} C_DIS
LIN {X 5.4565,Y -5.2226,Z 45,A -2.6892,B 0,C 0,E1 0.1598,E2 90.0718} C_DIS
LIN {X 5.9738,Y -4.6212,Z 45,A -2.6445,B 0,C 0,E1 0.1598,E2 90.0718} C_DIS
LIN {X 6.5327,Y -3.8022,Z 45,A -2.5888,B 0,C 0,E1 0.1598,E2 90.0718} C_DIS
LIN {X 7.0354,Y -2.7446,Z 45,A -2.5249,B 0,C 0,E1 0.1598,E2 90.0716} C_DIS
LIN {X 7.298,Y -1.9445,Z 45,A -2.4813,B 0,C 0,E1 0.1598,E2 90.0719} C_DIS
LIN {X 7.5159,Y -0.7886,Z 45,A -2.4237,B 0,C 0,E1 0.1598,E2 90.0716} C_DIS
LIN {X 7.5556,Y 0.1436,Z 45,A -2.3826,B 0,C 0,E1 0.1598,E2 90.0719} C_DIS
LIN {X 7.4538,Y 1.2441,Z 45,A -2.3391,B 0,C 0,E1 0.1598,E2 90.0717} C_DIS
LIN {X 7.1563,Y 2.4327,Z 45,A -2.2993,B 0,C 0,E1 0.1598,E2 90.0717} C_DIS
LIN {X 6.8017,Y 3.292,Z 45,A -2.276,B 0,C 0,E1 0.1598,E2 90.072} C_DIS
LIN {X 6.1375,Y 4.4101,Z 45,A -2.2526,B 0,C 0,E1 0.1598,E2 90.0718} C_DIS
LIN {X 5.3436,Y 5.3381,Z 45,A -2.2425,B 0,C 0,E1 0.1598,E2 90.072} C_DIS
LIN {X 4.5226,Y 6.0545,Z 45,A -2.2425,B 0,C 0,E1 0.1598,E2 90.0722} C_DIS
LIN {X 3.7384,Y 6.5679,Z 45,A -2.2497,B 0,C 0,E1 0.1598,E2 90.0724} C_DIS
LIN {X 2.5981,Y 7.0959,Z 45,A -2.2694,B 0,C 0,E1 0.1598,E2 90.0724} C_DIS
LIN {X 1.3698,Y 7.4334,Z 45,A -2.3004,B 0,C 0,E1 0.1598,E2 90.0724} C_DIS
LIN {X 0.4673,Y 7.5426,Z 45,A -2.3292,B 0,C 0,E1 0.1598,E2 90.0724} C_DIS
LIN {X -0.6977,Y 7.5262,Z 45,A -2.3729,B 0,C 0,E1 0.1598,E2 90.0724} C_DIS
LIN {X -1.5419,Y 7.3978,Z 45,A -2.4095,B 0,C 0,E1 0.1598,E2 90.0724} C_DIS
LIN {X -2.5705,Y 7.1061,Z 45,A -2.4598,B 0,C 0,E1 0.1598,E2 90.0723} C_DIS
LIN {X -3.8249,Y 6.5181,Z 45,A -2.5308,B 0,C 0,E1 0.1598,E2 90.072} C_DIS
LIN {X -4.6063,Y 5.9901,Z 45,A -2.582,B 0,C 0,E1 0.1598,E2 90.072} C_DIS
LIN {X -5.4408,Y 5.2383,Z 45,A -2.6445,B 0,C 0,E1 0.1598,E2 90.0717} C_DIS
LIN {X -6.0791,Y 4.4907,Z 45,A -2.6996,B 0,C 0,E1 0.1598,E2 90.0717} C_DIS
LIN {X -6.6861,Y 3.5126,Z 45,A -2.7631,B 0,C 0,E1 0.1598,E2 90.0713} C_DIS
LIN {X -7.119,Y 2.5352,Z 45,A -2.8204,B 0,C 0,E1 0.1598,E2 90.0713} C_DIS
LIN {X -7.4105,Y 1.4813,Z 45,A -2.8757,B 0,C 0,E1 0.1598,E2 90.0711} C_DIS
LIN {X -7.5383,Y 0.53,Z 45,A -2.9208,B 0,C 0,E1 0.1598,E2 90.0712} C_DIS
LIN {X -7.5352,Y -0.5759,Z 45,A -2.9673,B 0,C 0,E1 0.1598,E2 90.071} C_DIS
LIN {X -7.3751,Y -1.6348,Z 45,A -3.0063,B 0,C 0,E1 0.1598,E2 90.071} C_DIS
LIN {X -7.1775,Y -2.3548,Z 45,A -3.0298,B 0,C 0,E1 0.1598,E2 90.0712} C_DIS
LIN {X -6.9096,Y -3.0518,Z 45,A -3.0495,B 0,C 0,E1 0.1598,E2 90.0712} C_DIS
LIN {X -6.5744,Y -3.7189,Z 45,A -3.0655,B 0,C 0,E1 0.1598,E2 90.0712} C_DIS
LIN {X -6.1747,Y -4.3495,Z 45,A -3.0776,B 0,C 0,E1 0.1598,E2 90.0712} C_DIS
LIN {X -5.7147,Y -4.9375,Z 45,A -3.0857,B 0,C 0,E1 0.1598,E2 90.0712} C_DIS
LIN {X -5.0666,Y -5.609,Z 45,A -3.0903,B 0,C 0,E1 0.1598,E2 90.0712} C_DIS
LIN {X -4.1533,Y -6.3078,Z 45,A -3.0865,B 0,C 0,E1 0.1598,E2 90.0712} C_DIS
LIN {X -3.4296,Y -6.7297,Z 45,A -3.078,B 0,C 0,E1 0.1598,E2 90.0714} C_DIS
LIN {X -2.35,Y -7.1826,Z 45,A -3.0577,B 0,C 0,E1 0.1598,E2 90.0714} C_DIS
LIN {X -1.2902,Y -7.4464,Z 45,A -3.0301,B 0,C 0,E1 0.1598,E2 90.0714} C_DIS
LIN {X -0.319,Y -7.5517,Z 45,A -2.999,B 0,C 0,E1 0.1598,E2 90.0716} C_DIS
LIN {X -0.319,Y -7.5517,Z 45,A -2.999,B 0,C 0,E1 0.1598,E2 90.0716} C_DIS
Enddeposition()
LIN {X -0.1049,Y -8.4884,Z 45,A -3.0301,B 0,C 0,E1 0.1598,E2 90.0703} C_DIS
Startdeposition()
$VEL.CP = VEL_PRINT
LIN {X -1.1138,Y -8.4185,Z 45,A -3.0652,B 0,C 0,E1 0.1598,E2 90.0714} C_DIS
LIN {X -2.3189,Y -8.1645,Z 45,A -3.0986,B 0,C 0,E1 0.1598,E2 90.0714} C_DIS
LIN {X -3.1332,Y -7.8877,Z 45,A -3.1167,B 0,C 0,E1 0.1598,E2 90.0714} C_DIS
LIN {X -3.9153,Y -7.5299,Z 45,A -3.1301,B 0,C 0,E1 0.1598,E2 90.0714} C_DIS
LIN {X -4.6572,Y -7.0949,Z 45,A -3.1388,B 0,C 0,E1 0.1598,E2 90.0713} C_DIS
LIN {X -5.3513,Y -6.5871,Z 45,A -3.1426,B 0,C 0,E1 0.1598,E2 90.0713} C_DIS
LIN {X -5.9905,Y -6.0116,Z 45,A -3.1416,B 0,C 0,E1 0.1598,E2 90.0713} C_DIS
LIN {X -6.5682,Y -5.3746,Z 45,A -3.1357,B 0,C 0,E1 0.1598,E2 90.0712} C_DIS
LIN {X -7.0785,Y -4.6823,Z 45,A -3.1251,B 0,C 0,E1 0.1598,E2 90.0712} C_DIS
LIN {X -7.5163,Y -3.9419,Z 45,A -3.1097,B 0,C 0,E1 0.1598,E2 90.0712} C_DIS
LIN {X -7.8766,Y -3.161,Z 45,A -3.0898,B 0,C 0,E1 0.1598,E2 90.0712} C_DIS
LIN {X -8.1559,Y -2.3476,Z 45,A -3.0656,B 0,C 0,E1 0.1598,E2 90.0712} C_DIS
LIN {X -8.3516,Y -1.5101,Z 45,A -3.0373,B 0,C 0,E1 0.1598,E2 90.0712} C_DIS
LIN {X -8.4799,Y -0.4428,Z 45,A -2.9966,B 0,C 0,E1 0.1598,E2 90.0709} C_DIS
LIN {X -8.4673,Y 0.6308,Z 45,A -2.9508,B 0,C 0,E1 0.1598,E2 90.071} C_DIS
LIN {X -8.3362,Y 1.6157,Z 45,A -2.9044,B 0,C 0,E1 0.1598,E2 90.0712} C_DIS
LIN {X -8.0279,Y 2.7531,Z 45,A -2.8447,B 0,C 0,E1 0.1598,E2 90.0711} C_DIS
LIN {X -7.6991,Y 3.5702,Z 45,A -2.7984,B 0,C 0,E1 0.1598,E2 90.0715} C_DIS
LIN {X -7.288,Y 4.3491,Z 45,A -2.7503,B 0,C 0,E1 0.1598,E2 90.0715} C_DIS
LIN {X -6.6667,Y 5.2579,Z 45,A -2.6888,B 0,C 0,E1 0.1598,E2 90.0715} C_DIS
LIN {X -5.9342,Y 6.0729,Z 45,A -2.6275,B 0,C 0,E1 0.1598,E2 90.0717} C_DIS
LIN {X -5.1356,Y 6.7563,Z 45,A -2.5692,B 0,C 0,E1 0.1598,E2 90.0719} C_DIS
LIN {X -4.4416,Y 7.2309,Z 45,A -2.5236,B 0,C 0,E1 0.1598,E2 90.0721} C_DIS
LIN {X -3.7041,Y 7.6347,Z 45,A -2.4794,B 0,C 0,E1 0.1598,E2 90.0721} C_DIS
LIN {X -2.7343,Y 8.04,Z 45,A -2.4264,B 0,C 0,E1 0.1598,E2 90.0722} C_DIS
LIN {X -1.4781,Y 8.3575,Z 45,A -2.3666,B 0,C 0,E1 0.1598,E2 90.0724} C_DIS
LIN {X -0.718,Y 8.4614,Z 45,A -2.3342,B 0,C 0,E1 0.1598,E2 90.0724} C_DIS
LIN {X 0.4475,Y 8.4755,Z 45,A -2.2905,B 0,C 0,E1 0.1598,E2 90.0725} C_DIS
LIN {X 1.2982,Y 8.3866,Z 45,A -2.2629,B 0,C 0,E1 0.1598,E2 90.0725} C_DIS
LIN {X 2.1357,Y 8.2122,Z 45,A -2.2394,B 0,C 0,E1 0.1598,E2 90.0725} C_DIS
LIN {X 2.9515,Y 7.9551,Z 45,A -2.2201,B 0,C 0,E1 0.1598,E2 90.0725} C_DIS
LIN {X 3.7372,Y 7.617,Z 45,A -2.2055,B 0,C 0,E1 0.1598,E2 90.0725} C_DIS
LIN {X 4.8178,Y 6.9906,Z 45,A -2.1921,B 0,C 0,E1 0.1598,E2 90.0724} C_DIS
LIN {X 5.7085,Y 6.2798,Z 45,A -2.1894,B 0,C 0,E1 0.1598,E2 90.0724} C_DIS
LIN {X 6.5011,Y 5.4609,Z 45,A -2.1949,B 0,C 0,E1 0.1598,E2 90.0722} C_DIS
LIN {X 7.2258,Y 4.4537,Z 45,A -2.2109,B 0,C 0,E1 0.1598,E2 90.072} C_DIS
LIN {X 7.642,Y 3.6904,Z 45,A -2.2284,B 0,C 0,E1 0.1598,E2 90.0722} C_DIS
LIN {X 7.9793,Y 2.8892,Z 45,A -2.2501,B 0,C 0,E1 0.1598,E2 90.0722} C_DIS
LIN {X 8.2328,Y 2.0577,Z 45,A -2.2763,B 0,C 0,E1 0.1598,E2 90.0722} C_DIS
LIN {X 8.4327,Y 0.9895,Z 45,A -2.3142,B 0,C 0,E1 0.1598,E2 90.0717} C_DIS
LIN {X 8.485,Y -0.3451,Z 45,A -2.3688,B 0,C 0,E1 0.1598,E2 90.0712} C_DIS
LIN {X 8.3557,Y -1.4919,Z 45,A -2.4229,B 0,C 0,E1 0.1598,E2 90.0715} C_DIS
LIN {X 8.1631,Y -2.3243,Z 45,A -2.4659,B 0,C 0,E1 0.1598,E2 90.0719} C_DIS
LIN {X 7.888,Y -3.1331,Z 45,A -2.5106,B 0,C 0,E1 0.1598,E2 90.0719} C_DIS
LIN {X 7.4345,Y -4.0999,Z 45,A -2.5684,B 0,C 0,E1 0.1598,E2 90.0716} C_DIS
LIN {X 6.7315,Y -5.1737,Z 45,A -2.64,B 0,C 0,E1 0.1598,E2 90.0715} C_DIS
LIN {X 6.0444,Y -5.9574,Z 45,A -2.699,B 0,C 0,E1 0.1598,E2 90.0717} C_DIS
LIN {X 5.4304,Y -6.5215,Z 45,A -2.7457,B 0,C 0,E1 0.1598,E2 90.0717} C_DIS
LIN {X 4.7641,Y -7.0227,Z 45,A -2.7916,B 0,C 0,E1 0.1598,E2 90.0717} C_DIS
LIN {X 4.0519,Y -7.4561,Z 45,A -2.8362,B 0,C 0,E1 0.1598,E2 90.0717} C_DIS
LIN {X 3.3007,Y -7.8174,Z 45,A -2.8792,B 0,C 0,E1 0.1598,E2 90.0717} C_DIS
LIN {X 2.1506,Y -8.2134,Z 45,A -2.9383,B 0,C 0,E1 0.1598,E2 90.0716} C_DIS
LIN {X 1.2198,Y -8.3982,Z 45,A -2.9803,B 0,C 0,E1 0.1598,E2 90.0716} C_DIS
LIN {X 0.4644,Y -8.4737,Z 45,A -3.0112,B 0,C 0,E1 0.1598,E2 90.0716} C_DIS
LIN {X 0.4644,Y -8.4737,Z 45,A -3.0112,B 0,C 0,E1 0.1598,E2 90.0716} C_DIS
Enddeposition()
LIN {X 0.0009,Y -4.7546,Z 46,A -2.8553,B 0,C 0,E1 0.1598,E2 90.0604} C_DIS
Startdeposition()
$VEL.CP = VEL_PRINT
LIN {X 0.0009,Y -4.7546,Z 46,A -2.861,B 0,C 0,E1 0.1598,E2 90.0661} C_DIS
LIN {X 0.8351,Y -4.6773,Z 46,A -2.832,B 0,C 0,E1 0.1598,E2 90.0711} C_DIS
LIN {X 1.4849,Y -4.5131,Z 46,A -2.8018,B 0,C 0,E1 0.1598,E2 90.0718} C_DIS
LIN {X 2.1052,Y -4.2591,Z 46,A -2.7682,B 0,C 0,E1 0.1598,E2 90.0718} C_DIS
LIN {X 2.8187,Y -3.8211,Z 46,A -2.7233,B 0,C 0,E1 0.1598,E2 90.0718} C_DIS
LIN {X 3.2093,Y -3.5044,Z 46,A -2.6955,B 0,C 0,E1 0.1598,E2 90.0719} C_DIS
LIN {X 3.6687,Y -3.0164,Z 46,A -2.6577,B 0,C 0,E1 0.1598,E2 90.0719} C_DIS
LIN {X 4.0574,Y -2.4704,Z 46,A -2.6202,B 0,C 0,E1 0.1598,E2 90.0719} C_DIS
LIN {X 4.3653,Y -1.8752,Z 46,A -2.5834,B 0,C 0,E1 0.1598,E2 90.0719} C_DIS
LIN {X 4.5859,Y -1.2423,Z 46,A -2.5483,B 0,C 0,E1 0.1598,E2 90.0719} C_DIS
LIN {X 4.7147,Y -0.5845,Z 46,A -2.5155,B 0,C 0,E1 0.1598,E2 90.0719} C_DIS
LIN {X 4.7516,Y 0.0847,Z 46,A -2.4856,B 0,C 0,E1 0.1598,E2 90.072} C_DIS
LIN {X 4.6925,Y 0.7526,Z 46,A -2.4593,B 0,C 0,E1 0.1598,E2 90.072} C_DIS
LIN {X 4.5404,Y 1.4055,Z 46,A -2.4371,B 0,C 0,E1 0.1598,E2 90.072} C_DIS
LIN {X 4.2972,Y 2.0303,Z 46,A -2.4194,B 0,C 0,E1 0.1598,E2 90.0721} C_DIS
LIN {X 3.9678,Y 2.6142,Z 46,A -2.4067,B 0,C 0,E1 0.1598,E2 90.0721} C_DIS
LIN {X 3.5602,Y 3.1464,Z 46,A -2.3991,B 0,C 0,E1 0.1598,E2 90.0722} C_DIS
LIN {X 3.0814,Y 3.6155,Z 46,A -2.3968,B 0,C 0,E1 0.1598,E2 90.0722} C_DIS
LIN {X 2.5422,Y 4.0135,Z 46,A -2.3998,B 0,C 0,E1 0.1598,E2 90.0722} C_DIS
LIN {X 1.9515,Y 4.3303,Z 46,A -2.4081,B 0,C 0,E1 0.1598,E2 90.0722} C_DIS
LIN {X 1.323,Y 4.5627,Z 46,A -2.4214,B 0,C 0,E1 0.1598,E2 90.0723} C_DIS
LIN {X 0.6678,Y 4.7035,Z 46,A -2.4396,B 0,C 0,E1 0.1598,E2 90.0723} C_DIS
LIN {X -0.0007,Y 4.7507,Z 46,A -2.4623,B 0,C 0,E1 0.1598,E2 90.0723} C_DIS
LIN {X -0.6695,Y 4.705,Z 46,A -2.4889,B 0,C 0,E1 0.1598,E2 90.0723} C_DIS
LIN {X -1.3244,Y 4.5628,Z 46,A -2.519,B 0,C 0,E1 0.1598,E2 90.0723} C_DIS
LIN {X -1.9541,Y 4.3323,Z 46,A -2.552,B 0,C 0,E1 0.1598,E2 90.0721} C_DIS
LIN {X -2.5441,Y 4.0139,Z 46,A -2.5872,B 0,C 0,E1 0.1598,E2 90.0721} C_DIS
LIN {X -3.0839,Y 3.6162,Z 46,A -2.6239,B 0,C 0,E1 0.1598,E2 90.072} C_DIS
LIN {X -3.5616,Y 3.1457,Z 46,A -2.6615,B 0,C 0,E1 0.1598,E2 90.072} C_DIS
LIN {X -3.9687,Y 2.6131,Z 46,A -2.699,B 0,C 0,E1 0.1598,E2 90.0718} C_DIS
LIN {X -4.2976,Y 2.0289,Z 46,A -2.7358,B 0,C 0,E1 0.1598,E2 90.0718} C_DIS
LIN {X -4.5375,Y 1.4029,Z 46,A -2.7712,B 0,C 0,E1 0.1598,E2 90.0717} C_DIS
LIN {X -4.6908,Y 0.7506,Z 46,A -2.8044,B 0,C 0,E1 0.1598,E2 90.0717} C_DIS
LIN {X -4.7513,Y 0.0831,Z 46,A -2.835,B 0,C 0,E1 0.1598,E2 90.0716} C_DIS
LIN {X -4.7022,Y -0.6693,Z 46,A -2.865,B 0,C 0,E1 0.1598,E2 90.0715} C_DIS
LIN {X -4.5609,Y -1.3242,Z 46,A -2.8876,B 0,C 0,E1 0.1598,E2 90.0715} C_DIS
LIN {X -4.3647,Y -1.877,Z 46,A -2.9039,B 0,C 0,E1 0.1598,E2 90.0715} C_DIS
LIN {X -4.0565,Y -2.4722,Z 46,A -2.9178,B 0,C 0,E1 0.1598,E2 90.0715} C_DIS
LIN {X -3.6682,Y -3.0186,Z 46,A -2.9268,B 0,C 0,E1 0.1598,E2 90.0715} C_DIS
LIN {X -3.2073,Y -3.5053,Z 46,A -2.9306,B 0,C 0,E1 0.1598,E2 90.0715} C_DIS
LIN {X -2.6822,Y -3.922,Z 46,A -2.929,B 0,C 0,E1 0.1598,E2 90.0715} C_DIS
LIN {X -2.104,Y -4.2612,Z 46,A -2.9222,B 0,C 0,E1 0.1598,E2 90.0716} C_DIS
LIN {X -1.4837,Y -4.5156,Z 46,A -2.9103,B 0,C 0,E1 0.1598,E2 90.0716} C_DIS
LIN {X -0.8335,Y -4.6792,Z 46,A -2.8934,B 0,C 0,E1 0.1598,E2 90.0716} C_DIS
LIN {X 0.0009,Y -4.7546,Z 46,A -2.866,B 0,C 0,E1 0.1598,E2 90.0717} C_DIS
Enddeposition()
LIN {X 0.0009,Y -4.7546,Z 46,A -2.866,B 0,C 0,E1 0.1598,E2 90.0717} C_DIS
Startdeposition()
$VEL.CP = VEL_PRINT
LIN {X -0.6345,Y -5.6492,Z 46,A -2.927,B 0,C 0,E1 0.1598,E2 90.0711} C_DIS
LIN {X -1.4165,Y -5.507,Z 46,A -2.9501,B 0,C 0,E1 0.1598,E2 90.0716} C_DIS
LIN {X -2.1689,Y -5.2513,Z 46,A -2.9669,B 0,C 0,E1 0.1598,E2 90.0716} C_DIS
LIN {X -2.8809,Y -4.899,Z 46,A -2.978,B 0,C 0,E1 0.1598,E2 90.0716} C_DIS
LIN {X -3.5375,Y -4.4512,Z 46,A -2.983,B 0,C 0,E1 0.1598,E2 90.0715} C_DIS
LIN {X -4.123,Y -3.9136,Z 46,A -2.9816,B 0,C 0,E1 0.1598,E2 90.0715} C_DIS
LIN {X -4.6293,Y -3.3008,Z 46,A -2.9742,B 0,C 0,E1 0.1598,E2 90.0714} C_DIS
LIN {X -5.0432,Y -2.6222,Z 46,A -2.9605,B 0,C 0,E1 0.1598,E2 90.0714} C_DIS
LIN {X -5.3588,Y -1.893,Z 46,A -2.9412,B 0,C 0,E1 0.1598,E2 90.0714} C_DIS
LIN {X -5.5706,Y -1.1272,Z 46,A -2.9165,B 0,C 0,E1 0.1598,E2 90.0714} C_DIS
LIN {X -5.6723,Y -0.3393,Z 46,A -2.8868,B 0,C 0,E1 0.1598,E2 90.0714} C_DIS
LIN {X -5.6397,Y 0.7613,Z 46,A -2.8387,B 0,C 0,E1 0.1598,E2 90.0712} C_DIS
LIN {X -5.4115,Y 1.7365,Z 46,A -2.7891,B 0,C 0,E1 0.1598,E2 90.0714} C_DIS
LIN {X -5.1129,Y 2.4798,Z 46,A -2.7468,B 0,C 0,E1 0.1598,E2 90.0716} C_DIS
LIN {X -4.7145,Y 3.1746,Z 46,A -2.7027,B 0,C 0,E1 0.1598,E2 90.0717} C_DIS
LIN {X -4.2209,Y 3.8055,Z 46,A -2.6578,B 0,C 0,E1 0.1598,E2 90.0718} C_DIS
LIN {X -3.6438,Y 4.3611,Z 46,A -2.6131,B 0,C 0,E1 0.1598,E2 90.0719} C_DIS
LIN {X -2.9938,Y 4.8289,Z 46,A -2.5693,B 0,C 0,E1 0.1598,E2 90.072} C_DIS
LIN {X -2.2858,Y 5.2033,Z 46,A -2.5274,B 0,C 0,E1 0.1598,E2 90.0721} C_DIS
LIN {X -1.5317,Y 5.4733,Z 46,A -2.4882,B 0,C 0,E1 0.1598,E2 90.0722} C_DIS
LIN {X -0.7471,Y 5.6349,Z 46,A -2.4524,B 0,C 0,E1 0.1598,E2 90.0722} C_DIS
LIN {X 0.0526,Y 5.6855,Z 46,A -2.4208,B 0,C 0,E1 0.1598,E2 90.0723} C_DIS
LIN {X 0.8512,Y 5.6204,Z 46,A -2.3941,B 0,C 0,E1 0.1598,E2 90.0723} C_DIS
LIN {X 1.6329,Y 5.4448,Z 46,A -2.3727,B 0,C 0,E1 0.1598,E2 90.0723} C_DIS
LIN {X 2.3817,Y 5.1599,Z 46,A -2.3572,B 0,C 0,E1 0.1598,E2 90.0723} C_DIS
LIN {X 3.0834,Y 4.7736,Z 46,A -2.3477,B 0,C 0,E1 0.1598,E2 90.0723} C_DIS
LIN {X 3.7248,Y 4.2939,Z 46,A -2.3444,B 0,C 0,E1 0.1598,E2 90.0723} C_DIS
LIN {X 4.2906,Y 3.7266,Z 46,A -2.3476,B 0,C 0,E1 0.1598,E2 90.0723} C_DIS
LIN {X 4.7714,Y 3.0861,Z 46,A -2.3572,B 0,C 0,E1 0.1598,E2 90.0722} C_DIS
LIN {X 5.1583,Y 2.3848,Z 46,A -2.3727,B 0,C 0,E1 0.1598,E2 90.0722} C_DIS
LIN {X 5.4437,Y 1.6363,Z 46,A -2.3941,B 0,C 0,E1 0.1598,E2 90.072} C_DIS
LIN {X 5.6203,Y 0.8549,Z 46,A -2.4209,B 0,C 0,E1 0.1598,E2 90.072} C_DIS
LIN {X 5.6861,Y 0.0564,Z 46,A -2.4525,B 0,C 0,E1 0.1598,E2 90.072} C_DIS
LIN {X 5.6518,Y -0.6553,Z 46,A -2.484,B 0,C 0,E1 0.1598,E2 90.0718} C_DIS
LIN {X 5.4594,Y -1.5793,Z 46,A -2.5305,B 0,C 0,E1 0.1598,E2 90.0718} C_DIS
LIN {X 5.205,Y -2.2903,Z 46,A -2.5703,B 0,C 0,E1 0.1598,E2 90.0718} C_DIS
LIN {X 4.8549,Y -2.9597,Z 46,A -2.6118,B 0,C 0,E1 0.1598,E2 90.0718} C_DIS
LIN {X 4.4195,Y -3.5767,Z 46,A -2.6541,B 0,C 0,E1 0.1598,E2 90.0718} C_DIS
LIN {X 3.9046,Y -4.129,Z 46,A -2.6966,B 0,C 0,E1 0.1598,E2 90.0718} C_DIS
LIN {X 3.3234,Y -4.6109,Z 46,A -2.7386,B 0,C 0,E1 0.1598,E2 90.0718} C_DIS
LIN {X 2.6837,Y -5.0121,Z 46,A -2.7792,B 0,C 0,E1 0.1598,E2 90.0718} C_DIS
LIN {X 1.9952,Y -5.3226,Z 46,A -2.8177,B 0,C 0,E1 0.1598,E2 90.0718} C_DIS
LIN {X 1.272,Y -5.5392,Z 46,A -2.8535,B 0,C 0,E1 0.1598,E2 90.0718} C_DIS
LIN {X 0.5266,Y -5.6589,Z 46,A -2.886,B 0,C 0,E1 0.1598,E2 90.0718} C_DIS
LIN {X 0.5266,Y -5.6589,Z 46,A -2.886,B 0,C 0,E1 0.1598,E2 90.0718} C_DIS
Enddeposition()
LIN {X -0.0677,Y -6.6205,Z 46,A -2.9477,B 0,C 0,E1 0.1598,E2 90.0705} C_DIS
Startdeposition()
$VEL.CP = VEL_PRINT
LIN {X 0.7969,Y -6.5716,Z 46,A -2.915,B 0,C 0,E1 0.1598,E2 90.0716} C_DIS
LIN {X 1.4796,Y -6.4533,Z 46,A -2.885,B 0,C 0,E1 0.1598,E2 90.0717} C_DIS
LIN {X 2.146,Y -6.2633,Z 46,A -2.8524,B 0,C 0,E1 0.1598,E2 90.0717} C_DIS
LIN {X 2.7885,Y -6.0041,Z 46,A -2.8178,B 0,C 0,E1 0.1598,E2 90.0717} C_DIS
LIN {X 3.4006,Y -5.6792,Z 46,A -2.7815,B 0,C 0,E1 0.1598,E2 90.0718} C_DIS
LIN {X 3.9766,Y -5.294,Z 46,A -2.7439,B 0,C 0,E1 0.1598,E2 90.0718} C_DIS
LIN {X 4.5082,Y -4.8495,Z 46,A -2.7054,B 0,C 0,E1 0.1598,E2 90.0718} C_DIS
LIN {X 4.9904,Y -4.3519,Z 46,A -2.6664,B 0,C 0,E1 0.1598,E2 90.0718} C_DIS
LIN {X 5.4165,Y -3.8054,Z 46,A -2.6274,B 0,C 0,E1 0.1598,E2 90.0719} C_DIS
LIN {X 5.7849,Y -3.2185,Z 46,A -2.5888,B 0,C 0,E1 0.1598,E2 90.0719} C_DIS
LIN {X 6.0901,Y -2.5964,Z 46,A -2.551,B 0,C 0,E1 0.1598,E2 90.0719} C_DIS
LIN {X 6.3281,Y -1.9456,Z 46,A -2.5145,B 0,C 0,E1 0.1598,E2 90.0719} C_DIS
LIN {X 6.4947,Y -1.273,Z 46,A -2.4796,B 0,C 0,E1 0.1598,E2 90.072} C_DIS
LIN {X 6.5937,Y -0.5873,Z 46,A -2.4467,B 0,C 0,E1 0.1598,E2 90.072} C_DIS
LIN {X 6.6183,Y 0.1052,Z 46,A -2.4162,B 0,C 0,E1 0.1598,E2 90.072} C_DIS
LIN {X 6.5735,Y 0.7967,Z 46,A -2.3884,B 0,C 0,E1 0.1598,E2 90.0721} C_DIS
LIN {X 6.4527,Y 1.4791,Z 46,A -2.3637,B 0,C 0,E1 0.1598,E2 90.0721} C_DIS
LIN {X 6.2628,Y 2.1456,Z 46,A -2.3423,B 0,C 0,E1 0.1598,E2 90.0721} C_DIS
LIN {X 6.0038,Y 2.7884,Z 46,A -2.3244,B 0,C 0,E1 0.1598,E2 90.0722} C_DIS
LIN {X 5.6806,Y 3.4012,Z 46,A -2.3102,B 0,C 0,E1 0.1598,E2 90.0722} C_DIS
LIN {X 5.292,Y 3.9748,Z 46,A -2.3001,B 0,C 0,E1 0.1598,E2 90.0723} C_DIS
LIN {X 4.8474,Y 4.5062,Z 46,A -2.2939,B 0,C 0,E1 0.1598,E2 90.0723} C_DIS
LIN {X 4.35,Y 4.9887,Z 46,A -2.2917,B 0,C 0,E1 0.1598,E2 90.0723} C_DIS
LIN {X 3.8044,Y 5.4158,Z 46,A -2.2937,B 0,C 0,E1 0.1598,E2 90.0723} C_DIS
LIN {X 3.2175,Y 5.7841,Z 46,A -2.2997,B 0,C 0,E1 0.1598,E2 90.0724} C_DIS
LIN {X 2.5955,Y 6.0895,Z 46,A -2.3097,B 0,C 0,E1 0.1598,E2 90.0724} C_DIS
LIN {X 1.9455,Y 6.3296,Z 46,A -2.3235,B 0,C 0,E1 0.1598,E2 90.0724} C_DIS
LIN {X 1.2732,Y 6.4977,Z 46,A -2.3412,B 0,C 0,E1 0.1598,E2 90.0724} C_DIS
LIN {X 0.587,Y 6.5941,Z 46,A -2.3624,B 0,C 0,E1 0.1598,E2 90.0724} C_DIS
LIN {X -0.1055,Y 6.6205,Z 46,A -2.3868,B 0,C 0,E1 0.1598,E2 90.0724} C_DIS
LIN {X -0.7969,Y 6.5735,Z 46,A -2.4143,B 0,C 0,E1 0.1598,E2 90.0724} C_DIS
LIN {X -1.4792,Y 6.4525,Z 46,A -2.4446,B 0,C 0,E1 0.1598,E2 90.0724} C_DIS
LIN {X -2.1458,Y 6.263,Z 46,A -2.4772,B 0,C 0,E1 0.1598,E2 90.0723} C_DIS
LIN {X -2.7877,Y 6.0017,Z 46,A -2.512,B 0,C 0,E1 0.1598,E2 90.0722} C_DIS
LIN {X -3.4008,Y 5.6791,Z 46,A -2.5482,B 0,C 0,E1 0.1598,E2 90.0722} C_DIS
LIN {X -3.9759,Y 5.2925,Z 46,A -2.5858,B 0,C 0,E1 0.1598,E2 90.072} C_DIS
LIN {X -4.5073,Y 4.8479,Z 46,A -2.6242,B 0,C 0,E1 0.1598,E2 90.072} C_DIS
LIN {X -4.9908,Y 4.3515,Z 46,A -2.663,B 0,C 0,E1 0.1598,E2 90.0719} C_DIS
LIN {X -5.4168,Y 3.805,Z 46,A -2.7018,B 0,C 0,E1 0.1598,E2 90.0719} C_DIS
LIN {X -5.7852,Y 3.2181,Z 46,A -2.7402,B 0,C 0,E1 0.1598,E2 90.0717} C_DIS
LIN {X -6.0881,Y 2.5949,Z 46,A -2.7777,B 0,C 0,E1 0.1598,E2 90.0717} C_DIS
LIN {X -6.3273,Y 1.9446,Z 46,A -2.8141,B 0,C 0,E1 0.1598,E2 90.0716} C_DIS
LIN {X -6.4957,Y 1.2725,Z 46,A -2.8487,B 0,C 0,E1 0.1598,E2 90.0716} C_DIS
LIN {X -6.5921,Y 0.5863,Z 46,A -2.8813,B 0,C 0,E1 0.1598,E2 90.0715} C_DIS
LIN {X -6.6192,Y -0.1059,Z 46,A -2.9116,B 0,C 0,E1 0.1598,E2 90.0715} C_DIS
LIN {X -6.5714,Y -0.7973,Z 46,A -2.9391,B 0,C 0,E1 0.1598,E2 90.0715} C_DIS
LIN {X -6.4532,Y -1.48,Z 46,A -2.9637,B 0,C 0,E1 0.1598,E2 90.0714} C_DIS
LIN {X -6.2628,Y -2.1462,Z 46,A -2.9849,B 0,C 0,E1 0.1598,E2 90.0714} C_DIS
LIN {X -6.0047,Y -2.7892,Z 46,A -3.0027,B 0,C 0,E1 0.1598,E2 90.0714} C_DIS
LIN {X -5.6791,Y -3.4008,Z 46,A -3.0167,B 0,C 0,E1 0.1598,E2 90.0714} C_DIS
LIN {X -5.2921,Y -3.9756,Z 46,A -3.0269,B 0,C 0,E1 0.1598,E2 90.0714} C_DIS
LIN {X -4.8476,Y -4.5071,Z 46,A -3.0332,B 0,C 0,E1 0.1598,E2 90.0714} C_DIS
LIN {X -4.3505,Y -4.99,Z 46,A -3.0355,B 0,C 0,E1 0.1598,E2 90.0714} C_DIS
LIN {X -3.8054,Y -5.4177,Z 46,A -3.0337,B 0,C 0,E1 0.1598,E2 90.0714} C_DIS
LIN {X -3.2178,Y -5.785,Z 46,A -3.0277,B 0,C 0,E1 0.1598,E2 90.0714} C_DIS
LIN {X -2.5965,Y -6.0919,Z 46,A -3.018,B 0,C 0,E1 0.1598,E2 90.0714} C_DIS
LIN {X -1.9456,Y -6.3298,Z 46,A -3.0043,B 0,C 0,E1 0.1598,E2 90.0715} C_DIS
LIN {X -1.2733,Y -6.4977,Z 46,A -2.9868,B 0,C 0,E1 0.1598,E2 90.0715} C_DIS
LIN {X -0.587,Y -6.5936,Z 46,A -2.9657,B 0,C 0,E1 0.1598,E2 90.0716} C_DIS
LIN {X -0.587,Y -6.5936,Z 46,A -2.9657,B 0,C 0,E1 0.1598,E2 90.0716} C_DIS
Enddeposition()
LIN {X -0.0679,Y -7.5518,Z 46,A -2.9865,B 0,C 0,E1 0.1598,E2 90.0704} C_DIS
Startdeposition()
$VEL.CP = VEL_PRINT
LIN {X -0.8518,Y -7.5087,Z 46,A -3.0145,B 0,C 0,E1 0.1598,E2 90.0715} C_DIS
LIN {X -1.8359,Y -7.3306,Z 46,A -3.043,B 0,C 0,E1 0.1598,E2 90.0715} C_DIS
LIN {X -2.8598,Y -6.9953,Z 46,A -3.0662,B 0,C 0,E1 0.1598,E2 90.0715} C_DIS
LIN {X -3.7997,Y -6.5273,Z 46,A -3.0808,B 0,C 0,E1 0.1598,E2 90.0714} C_DIS
LIN {X -4.6705,Y -5.9407,Z 46,A -3.0877,B 0,C 0,E1 0.1598,E2 90.0712} C_DIS
LIN {X -5.4627,Y -5.2152,Z 46,A -3.0859,B 0,C 0,E1 0.1598,E2 90.0712} C_DIS
LIN {X -5.951,Y -4.6499,Z 46,A -3.0799,B 0,C 0,E1 0.1598,E2 90.0712} C_DIS
LIN {X -6.3822,Y -4.04,Z 46,A -3.0699,B 0,C 0,E1 0.1598,E2 90.0712} C_DIS
LIN {X -6.7502,Y -3.3899,Z 46,A -3.0558,B 0,C 0,E1 0.1598,E2 90.0712} C_DIS
LIN {X -7.0522,Y -2.7066,Z 46,A -3.0379,B 0,C 0,E1 0.1598,E2 90.0712} C_DIS
LIN {X -7.2854,Y -1.9968,Z 46,A -3.0164,B 0,C 0,E1 0.1598,E2 90.0712} C_DIS
LIN {X -7.4797,Y -1.0834,Z 46,A -2.9846,B 0,C 0,E1 0.1598,E2 90.0711} C_DIS
LIN {X -7.5586,Y 0,Z 46,A -2.9415,B 0,C 0,E1 0.1598,E2 90.0711} C_DIS
LIN {X -7.4973,Y 0.952,Z 46,A -2.8991,B 0,C 0,E1 0.1598,E2 90.0712} C_DIS
LIN {X -7.2842,Y 2.0141,Z 46,A -2.8461,B 0,C 0,E1 0.1598,E2 90.0712} C_DIS
LIN {X -6.8747,Y 3.128,Z 46,A -2.7838,B 0,C 0,E1 0.1598,E2 90.0712} C_DIS
LIN {X -6.3695,Y 4.0672,Z 46,A -2.7256,B 0,C 0,E1 0.1598,E2 90.0714} C_DIS
LIN {X -5.7087,Y 4.9448,Z 46,A -2.6642,B 0,C 0,E1 0.1598,E2 90.0716} C_DIS
LIN {X -5.0216,Y 5.6483,Z 46,A -2.6092,B 0,C 0,E1 0.1598,E2 90.0718} C_DIS
LIN {X -4.1907,Y 6.2886,Z 46,A -2.5516,B 0,C 0,E1 0.1598,E2 90.072} C_DIS
LIN {X -3.2702,Y 6.8123,Z 46,A -2.4955,B 0,C 0,E1 0.1598,E2 90.072} C_DIS
LIN {X -2.088,Y 7.2645,Z 46,A -2.4328,B 0,C 0,E1 0.1598,E2 90.0722} C_DIS
LIN {X -0.909,Y 7.4996,Z 46,A -2.3793,B 0,C 0,E1 0.1598,E2 90.0724} C_DIS
LIN {X -0.1032,Y 7.5566,Z 46,A -2.3472,B 0,C 0,E1 0.1598,E2 90.0724} C_DIS
LIN {X 1.0496,Y 7.4851,Z 46,A -2.3077,B 0,C 0,E1 0.1598,E2 90.0724} C_DIS
LIN {X 1.8736,Y 7.3208,Z 46,A -2.2842,B 0,C 0,E1 0.1598,E2 90.0724} C_DIS
LIN {X 3.0815,Y 6.9011,Z 46,A -2.2574,B 0,C 0,E1 0.1598,E2 90.0724} C_DIS
LIN {X 4.0699,Y 6.3679,Z 46,A -2.2436,B 0,C 0,E1 0.1598,E2 90.0724} C_DIS
LIN {X 5.024,Y 5.6394,Z 46,A -2.2392,B 0,C 0,E1 0.1598,E2 90.0722} C_DIS
LIN {X 5.7854,Y 4.8614,Z 46,A -2.2442,B 0,C 0,E1 0.1598,E2 90.0722} C_DIS
LIN {X 6.4064,Y 4.0064,Z 46,A -2.2577,B 0,C 0,E1 0.1598,E2 90.0722} C_DIS
LIN {X 6.8006,Y 3.2944,Z 46,A -2.2736,B 0,C 0,E1 0.1598,E2 90.0722} C_DIS
LIN {X 7.1558,Y 2.4343,Z 46,A -2.2972,B 0,C 0,E1 0.1598,E2 90.0722} C_DIS
LIN {X 7.4538,Y 1.2445,Z 46,A -2.3365,B 0,C 0,E1 0.1598,E2 90.0716} C_DIS
LIN {X 7.5521,Y 0.302,Z 46,A -2.3735,B 0,C 0,E1 0.1598,E2 90.0719} C_DIS
LIN {X 7.5197,Y -0.7548,Z 46,A -2.4196,B 0,C 0,E1 0.1598,E2 90.0717} C_DIS
LIN {X 7.2972,Y -1.9478,Z 46,A -2.4786,B 0,C 0,E1 0.1598,E2 90.0715} C_DIS
LIN {X 7.0315,Y -2.7548,Z 46,A -2.5232,B 0,C 0,E1 0.1598,E2 90.0718} C_DIS
LIN {X 6.5224,Y -3.8193,Z 46,A -2.5872,B 0,C 0,E1 0.1598,E2 90.0716} C_DIS
LIN {X 6.0191,Y -4.565,Z 46,A -2.6378,B 0,C 0,E1 0.1598,E2 90.0718} C_DIS
LIN {X 5.4354,Y -5.2497,Z 46,A -2.6884,B 0,C 0,E1 0.1598,E2 90.0718} C_DIS
LIN {X 4.6469,Y -5.9556,Z 46,A -2.7475,B 0,C 0,E1 0.1598,E2 90.0717} C_DIS
LIN {X 4.041,Y -6.3819,Z 46,A -2.7881,B 0,C 0,E1 0.1598,E2 90.0717} C_DIS
LIN {X 3.2315,Y -6.8311,Z 46,A -2.8369,B 0,C 0,E1 0.1598,E2 90.0717} C_DIS
LIN {X 2.1457,Y -7.2465,Z 46,A -2.8945,B 0,C 0,E1 0.1598,E2 90.0717} C_DIS
LIN {X 1.2347,Y -7.4527,Z 46,A -2.9367,B 0,C 0,E1 0.1598,E2 90.0717} C_DIS
LIN {X 0.4925,Y -7.5389,Z 46,A -2.9676,B 0,C 0,E1 0.1598,E2 90.0717} C_DIS
LIN {X 0.4925,Y -7.5389,Z 46,A -2.9676,B 0,C 0,E1 0.1598,E2 90.0717} C_DIS
Enddeposition()
LIN {X -0.0867,Y -8.4896,Z 46,A -3.0284,B 0,C 0,E1 0.1598,E2 90.0703} C_DIS
Startdeposition()
$VEL.CP = VEL_PRINT
LIN {X 0.9367,Y -8.4334,Z 46,A -2.9896,B 0,C 0,E1 0.1598,E2 90.0715} C_DIS
LIN {X 1.7463,Y -8.3036,Z 46,A -2.9545,B 0,C 0,E1 0.1598,E2 90.0716} C_DIS
LIN {X 2.5398,Y -8.0968,Z 46,A -2.9166,B 0,C 0,E1 0.1598,E2 90.0716} C_DIS
LIN {X 3.3099,Y -7.815,Z 46,A -2.8763,B 0,C 0,E1 0.1598,E2 90.0717} C_DIS
LIN {X 4.3631,Y -7.2842,Z 46,A -2.8149,B 0,C 0,E1 0.1598,E2 90.0717} C_DIS
LIN {X 5.4885,Y -6.4775,Z 46,A -2.739,B 0,C 0,E1 0.1598,E2 90.0716} C_DIS
LIN {X 6.3173,Y -5.668,Z 46,A -2.674,B 0,C 0,E1 0.1598,E2 90.0716} C_DIS
LIN {X 6.8582,Y -4.9999,Z 46,A -2.6257,B 0,C 0,E1 0.1598,E2 90.0718} C_DIS
LIN {X 7.3287,Y -4.2805,Z 46,A -2.5777,B 0,C 0,E1 0.1598,E2 90.0718} C_DIS
LIN {X 7.7241,Y -3.5172,Z 46,A -2.5305,B 0,C 0,E1 0.1598,E2 90.0718} C_DIS
LIN {X 8.0402,Y -2.7179,Z 46,A -2.4847,B 0,C 0,E1 0.1598,E2 90.0719} C_DIS
LIN {X 8.2739,Y -1.8907,Z 46,A -2.4407,B 0,C 0,E1 0.1598,E2 90.0719} C_DIS
LIN {X 8.4231,Y -1.0441,Z 46,A -2.3991,B 0,C 0,E1 0.1598,E2 90.0719} C_DIS
LIN {X 8.4864,Y -0.1869,Z 46,A -2.3601,B 0,C 0,E1 0.1598,E2 90.072} C_DIS
LIN {X 8.4327,Y 0.9896,Z 46,A -2.3115,B 0,C 0,E1 0.1598,E2 90.0717} C_DIS
LIN {X 8.2326,Y 2.0582,Z 46,A -2.2733,B 0,C 0,E1 0.1598,E2 90.0719} C_DIS
LIN {X 7.9788,Y 2.8902,Z 46,A -2.2474,B 0,C 0,E1 0.1598,E2 90.0721} C_DIS
LIN {X 7.6412,Y 3.6918,Z 46,A -2.2256,B 0,C 0,E1 0.1598,E2 90.0722} C_DIS
LIN {X 7.2245,Y 4.4554,Z 46,A -2.2084,B 0,C 0,E1 0.1598,E2 90.0722} C_DIS
LIN {X 6.5023,Y 5.4596,Z 46,A -2.192,B 0,C 0,E1 0.1598,E2 90.0721} C_DIS
LIN {X 5.7104,Y 6.2782,Z 46,A -2.1866,B 0,C 0,E1 0.1598,E2 90.0723} C_DIS
LIN {X 4.8205,Y 6.9888,Z 46,A -2.1891,B 0,C 0,E1 0.1598,E2 90.0723} C_DIS
LIN {X 3.7499,Y 7.6111,Z 46,A -2.2023,B 0,C 0,E1 0.1598,E2 90.0723} C_DIS
LIN {X 2.9822,Y 7.944,Z 46,A -2.2166,B 0,C 0,E1 0.1598,E2 90.0725} C_DIS
LIN {X 2.1854,Y 8.1999,Z 46,A -2.2352,B 0,C 0,E1 0.1598,E2 90.0725} C_DIS
LIN {X 1.3674,Y 8.3768,Z 46,A -2.2579,B 0,C 0,E1 0.1598,E2 90.0725} C_DIS
LIN {X 0.2448,Y 8.4873,Z 46,A -2.2947,B 0,C 0,E1 0.1598,E2 90.0725} C_DIS
LIN {X -0.7184,Y 8.4614,Z 46,A -2.3314,B 0,C 0,E1 0.1598,E2 90.0725} C_DIS
LIN {X -1.9417,Y 8.262,Z 46,A -2.385,B 0,C 0,E1 0.1598,E2 90.0724} C_DIS
LIN {X -2.7332,Y 8.0404,Z 46,A -2.4236,B 0,C 0,E1 0.1598,E2 90.0724} C_DIS
LIN {X -3.7023,Y 7.6355,Z 46,A -2.4765,B 0,C 0,E1 0.1598,E2 90.0722} C_DIS
LIN {X -4.4393,Y 7.2323,Z 46,A -2.5207,B 0,C 0,E1 0.1598,E2 90.0722} C_DIS
LIN {X -5.1329,Y 6.7583,Z 46,A -2.5663,B 0,C 0,E1 0.1598,E2 90.072} C_DIS
LIN {X -5.9312,Y 6.0758,Z 46,A -2.6245,B 0,C 0,E1 0.1598,E2 90.0718} C_DIS
LIN {X -6.6741,Y 5.2483,Z 46,A -2.6868,B 0,C 0,E1 0.1598,E2 90.0716} C_DIS
LIN {X -7.2923,Y 4.3424,Z 46,A -2.7479,B 0,C 0,E1 0.1598,E2 90.0716} C_DIS
LIN {X -7.7013,Y 3.5661,Z 46,A -2.7959,B 0,C 0,E1 0.1598,E2 90.0716} C_DIS
LIN {X -8.0285,Y 2.7519,Z 46,A -2.8423,B 0,C 0,E1 0.1598,E2 90.0714} C_DIS
LIN {X -8.336,Y 1.617,Z 46,A -2.9014,B 0,C 0,E1 0.1598,E2 90.0711} C_DIS
LIN {X -8.4677,Y 0.6249,Z 46,A -2.9482,B 0,C 0,E1 0.1598,E2 90.0711} C_DIS
LIN {X -8.4797,Y -0.4466,Z 46,A -2.9939,B 0,C 0,E1 0.1598,E2 90.0709} C_DIS
LIN {X -8.3513,Y -1.5135,Z 46,A -3.0344,B 0,C 0,E1 0.1598,E2 90.0709} C_DIS
LIN {X -8.1554,Y -2.3506,Z 46,A -3.0628,B 0,C 0,E1 0.1598,E2 90.0711} C_DIS
LIN {X -7.8758,Y -3.1635,Z 46,A -3.087,B 0,C 0,E1 0.1598,E2 90.0711} C_DIS
LIN {X -7.5154,Y -3.944,Z 46,A -3.1069,B 0,C 0,E1 0.1598,E2 90.0711} C_DIS
LIN {X -7.0776,Y -4.6839,Z 46,A -3.1222,B 0,C 0,E1 0.1598,E2 90.0711} C_DIS
LIN {X -6.5674,Y -5.3758,Z 46,A -3.1328,B 0,C 0,E1 0.1598,E2 90.0711} C_DIS
LIN {X -5.9898,Y -6.0125,Z 46,A -3.1387,B 0,C 0,E1 0.1598,E2 90.0711} C_DIS
LIN {X -5.3508,Y -6.5876,Z 46,A -3.1397,B 0,C 0,E1 0.1598,E2 90.0712} C_DIS
Enddeposition()
END
